// Mitsubishi GX Works2 project: CV_B01-20251214_0   PLC: Q03UDV

TYPE DInput : STRUCT
  In_Power : BOOL;  (* 输入电源 *)
  X01_1 : BOOL;  (* X01_1 *)
  B01_Emergency_Stop_Circuit1 : BOOL;  (* BO1急停回路1 *)
  B01_Emergency_Stop_Circuit2 : BOOL;  (* BO1急停回路2 *)
  B01_Grating_Circuit1 : BOOL;  (* BO1光栅回路1 *)
  B01_Grating_Circuit2 : BOOL;  (* BO1光栅回路2 *)
  B01_Safety_Door_Circuit1 : BOOL;  (* BO1安全门回路1 *)
  B01_Safety_Door_Circuit2 : BOOL;  (* BO1安全门回路2 *)
  AO1Safety_Circuit1 : BOOL;  (* AO1急停回路1 *)
  AO1Safety_Circuit2 : BOOL;  (* AO1急停回路2 *)
  B02_Emergency_Stop_Circuit1 : BOOL;  (* BO2急停回路1 *)
  B02_Emergency_Stop_Circuit2 : BOOL;  (* BO2急停回路2 *)
  B02_Grating_Circuit1 : BOOL;  (* BO2光栅回路1 *)
  B02_Grating_Circuit2 : BOOL;  (* BO2光栅回路2 *)
  B02_Safety_Door_Circuit1 : BOOL;  (* BO2安全门回路1 *)
  B02_Safety_Door_Circuit2 : BOOL;  (* BO2安全门回路2 *)
  Manual_Auto : BOOL;  (* 手动自动 *)
  Single_OnLine : BOOL;  (* 单机联机 *)
  X02_2 : BOOL;  (* X02_2 *)
  Admin : BOOL;  (* 管理者 *)
  Alarm_Reset : BOOL;  (* 故障复位 *)
  Ready_Button : BOOL;  (* 就绪按钮 *)
  Start_Button : BOOL;  (* 启动按钮 *)
  Pause_Button : BOOL;  (* 暂停按钮 *)
  Lamp_Check : BOOL;  (* 灯光检查按钮 *)
  X09_2 : BOOL;  (* X09_2 *)
  Operational_Ready1 : BOOL;  (* 运行准备01 *)
  Operational_Ready2 : BOOL;  (* 运行准备02 *)
  Operational_Ready11 : BOOL;  (* 运行准备11 *)
  Operational_Ready12 : BOOL;  (* 运行准备12 *)
  Air_Error : BOOL;  (* 柜机空调故障 *)
  X0F_2 : BOOL;  (* X0F_2 *)
  CV01顶升上限检测 : BOOL;  (* CV01顶升上限检测 *)
  CV01顶升下限检测 : BOOL;  (* CV01顶升下限检测 *)
  CV01顶升故障检测 : BOOL;  (* CV01顶升故障检测 *)
  CV01顶升电源检测 : BOOL;  (* CV01顶升电源检测 *)
  CV01物料停止检测 : BOOL;  (* CV01物料停止检测 *)
  X05_3 : BOOL;  (* X05_3 *)
  CV01伸缩中位检测1 : BOOL;  (* CV01伸缩中位检测1 *)
  CV01伸缩中位检测2 : BOOL;  (* CV01伸缩中位检测2 *)
  CV01伸缩极限检测 : BOOL;  (* CV01伸缩极限检测 *)
  CV01伸缩电源检测 : BOOL;  (* CV01伸缩电源检测 *)
  CV01AGV物料检测 : BOOL;  (* CV01AGV物料检测 *)
  CV01AGV本体检测1 : BOOL;  (* CV01AGV本体检测1 *)
  CV01AGV本体检测2 : BOOL;  (* CV01AGV本体检测2 *)
  CV01超宽检测1 : BOOL;  (* CV01超宽检测1 *)
  CV01超宽检测2 : BOOL;  (* CV01超宽检测2 *)
  CV01超高检测 : BOOL;  (* CV01超高检测 *)
  Bx03顶升上限检测 : BOOL;  (* Bx03顶升上限检测 *)
  Bx03顶升下限检测 : BOOL;  (* Bx03顶升下限检测 *)
  Bx03顶升故障检测 : BOOL;  (* Bx03顶升故障检测 *)
  Bx03顶升电源检测 : BOOL;  (* Bx03顶升电源检测 *)
  Bx03物料停止检测 : BOOL;  (* Bx03物料停止检测 *)
  Bx03物料减速检测 : BOOL;  (* Bx03物料减速检测 *)
  CV02伸缩中位检测1 : BOOL;  (* Bx03伸缩中位检测1 *)
  CV02伸缩中位检测2 : BOOL;  (* Bx03伸缩中位检测2 *)
  CV02伸缩极限检测 : BOOL;  (* Bx03伸缩极限检测 *)
  Bx03伸缩电源检测 : BOOL;  (* Bx03伸缩电源检测 *)
  Bx03AGV物料检测 : BOOL;  (* Bx03AGV物料检测 *)
  Bx03AGV本体检测1 : BOOL;  (* Bx03AGV本体检测1 *)
  Bx03AGV本体检测2 : BOOL;  (* Bx03AGV本体检测2 *)
  X0D_4 : BOOL;  (* X0D_4 *)
  X0E_4 : BOOL;  (* X0E_4 *)
  X0F_4 : BOOL;  (* X0F_4 *)
  Bx02顶升上限检测 : BOOL;  (* Bx02顶升上限检测 *)
  Bx02顶升下限检测 : BOOL;  (* Bx02顶升下限检测 *)
  Bx02顶升故障检测 : BOOL;  (* Bx02顶升故障检测 *)
  Bx02顶升电源检测 : BOOL;  (* Bx02顶升电源检测 *)
  Bx02物料到位检测 : BOOL;  (* Bx02物料到位检测 *)
  Bx02物料减速检测 : BOOL;  (* Bx02物料减速检测 *)
  Bx02输送故障检测 : BOOL;  (* Bx02输送故障检测 *)
  Bx02输送电源检测 : BOOL;  (* Bx02输送电源检测 *)
  Bx04顶升上限检测 : BOOL;  (* Bx04顶升上限检测 *)
  Bx04顶升下限检测 : BOOL;  (* Bx04顶升下限检测 *)
  Bx04顶升故障检测 : BOOL;  (* Bx04顶升故障检测 *)
  Bx04顶升电源检测 : BOOL;  (* Bx04顶升电源检测 *)
  Bx04物料到位检测 : BOOL;  (* Bx04物料到位检测 *)
  X0D_5 : BOOL;  (* X0D_5 *)
  Bx04输送故障检测 : BOOL;  (* Bx04输送故障检测 *)
  Bx04输送电源检测 : BOOL;  (* Bx04输送电源检测 *)
  AGV侧安全光栅输入信号1 : BOOL;  (* AGV侧安全光栅输入信号1 *)
  AGV侧安全光栅输入信号2 : BOOL;  (* AGV侧安全光栅输入信号2 *)
  AGV侧安全光栅输入信号11 : BOOL;  (* AGV侧安全光栅输入信号11 *)
  AGV侧安全光栅输入信号12 : BOOL;  (* AGV侧安全光栅输入信号12 *)
  CV_IN侧安全光栅输入信号1 : BOOL;  (* CV_IN侧安全光栅输入信号1 *)
  CV_IN侧安全光栅输入信号2 : BOOL;  (* CV_IN侧安全光栅输入信号2 *)
  CV_Out侧安全光栅输入信号1 : BOOL;  (* CV_Out侧安全光栅输入信号1 *)
  CV_Out侧安全光栅输入信号2 : BOOL;  (* CV_Out侧安全光栅输入信号2 *)
  X08_6 : BOOL;  (* X08_6 *)
  X09_6 : BOOL;  (* X09_6 *)
  安全门1输入信号1 : BOOL;  (* 安全门1输入信号1 *)
  安全门1输入信号2 : BOOL;  (* 安全门1输入信号2 *)
  解锁1安全门 : BOOL;  (* 解锁1安全门 *)
  X0D_6 : BOOL;  (* X0D_6 *)
  X0E_6 : BOOL;  (* X0E_6 *)
  X0F_6 : BOOL;  (* X0F_6 *)
  Photonic1_output1 : BOOL;  (* Photonic1_output1 *)
  Photonic1_output2 : BOOL;  (* Photonic1_output2 *)
  Photonic1_output3 : BOOL;  (* Photonic1_output3 *)
  Photonic1_output4 : BOOL;  (* Photonic1_output4 *)
  Photonic1_Go : BOOL;  (* Photonic1_Go *)
  X05_7 : BOOL;  (* X05_7 *)
  Photonic2_output1 : BOOL;  (* Photonic2_output1 *)
  Photonic2_output2 : BOOL;  (* Photonic2_output2 *)
  Photonic2_output3 : BOOL;  (* Photonic2_output3 *)
  Photonic2_output4 : BOOL;  (* Photonic2_output4 *)
  Photonic2_Go : BOOL;  (* Photonic2_Go *)
  X0B_7 : BOOL;  (* X0B_7 *)
  Photonic3_output1 : BOOL;  (* Photonic3_output1 *)
  Photonic3_output2 : BOOL;  (* Photonic3_output2 *)
  Photonic3_output3 : BOOL;  (* Photonic3_output3 *)
  Photonic3_output4 : BOOL;  (* Photonic3_output4 *)
  Photonic3_Go : BOOL;  (* Photonic3_Go *)
  X01_8 : BOOL;  (* X01_8 *)
  Photonic4_output1 : BOOL;  (* Photonic4_output1 *)
  Photonic4_output2 : BOOL;  (* Photonic4_output2 *)
  Photonic4_output3 : BOOL;  (* Photonic4_output3 *)
  Photonic4_output4 : BOOL;  (* Photonic4_output4 *)
  Photonic4_Go : BOOL;  (* Photonic4_Go *)
  X07_8 : BOOL;  (* X07_8 *)
  X08_8 : BOOL;  (* X08_8 *)
  X09_8 : BOOL;  (* X09_8 *)
  X0A_8 : BOOL;  (* X0A_8 *)
  X0B_8 : BOOL;  (* X0B_8 *)
  X0C_8 : BOOL;  (* X0C_8 *)
  X0D_8 : BOOL;  (* X0D_8 *)
  X0E_8 : BOOL;  (* X0E_8 *)
  X0F_8 : BOOL;  (* X0F_8 *)
END_STRUCT END_TYPE

TYPE DOutput : STRUCT
  Pole_Light_R : BOOL;  (* 柜体灯_红 *)
  Pole_Light_Y : BOOL;  (* 柜体灯_黄 *)
  Pole_Light_G : BOOL;  (* 柜体灯_绿 *)
  HA01_Sound1 : BOOL;  (* 蜂鸣器通道1 *)
  HA01_Sound2 : BOOL;  (* 蜂鸣器通道2 *)
  HA01_Sound3 : BOOL;  (* 蜂鸣器通道3 *)
  HA01_Sound4 : BOOL;  (* 蜂鸣器通道4 *)
  Y07_1 : BOOL;  (* Y07_1 *)
  Ready_Button_Indicator_Light : BOOL;  (* 就绪按钮灯 *)
  Start_Button_Indicator_Light : BOOL;  (* 启动按钮灯 *)
  Pause_Button_Indicator_Light : BOOL;  (* 暂停按钮灯 *)
  Y0B_1 : BOOL;  (* Y0B_1 *)
  Y0C_1 : BOOL;  (* Y0C_1 *)
  Y0D_1 : BOOL;  (* Y0D_1 *)
  SafetyDoor_Indicator_Light : BOOL;  (* Lock the Safety Door *)
  Unlock_SafetyDoor : BOOL;  (* 解锁安全门 *)
  CV1_JackingUP_Fork_Run : BOOL;  (* Bx01顶升正转运行 *)
  CV1_JackingDown_Fork_Run : BOOL;  (* Bx01顶升反转运行 *)
  CV1_Jacking_Fork_Reset : BOOL;  (* Bx01顶升故障复位 *)
  Y03_2 : BOOL;  (* Y03_2 *)
  Grat1_Warning_Light_R : BOOL;  (* 光栅1警示灯_红 *)
  Grat1_Warning_Light_G : BOOL;  (* 光栅1警示灯_绿 *)
  CV1_JackingUP_Run : BOOL;  (* Bx02顶升正转运行 *)
  CV1_JackingDown_Run : BOOL;  (* Bx02顶升反转运行 *)
  CV1_Jacking_Reset : BOOL;  (* Bx02顶升故障复位 *)
  Y09_2 : BOOL;  (* Y09_2 *)
  CV1_ConveyingIN_Run : BOOL;  (* Bx02输送正转运行 *)
  CV1_ConveyingOut_Run : BOOL;  (* Bx02输送反转运行 *)
  CV1_Conveying_SpeedA : BOOL;  (* Bx02输送速度A *)
  CV1_Conveying_SpeedB : BOOL;  (* Bx02输送速度B *)
  CV1_Conveying_Reset : BOOL;  (* Bx02输送故障复位 *)
  Y0F_2 : BOOL;  (* Y0F_2 *)
  CV2_JackingUP_Fork_Run : BOOL;  (* Bx03顶升正转运行 *)
  CV2_JackingDown_Fork_Run : BOOL;  (* Bx03顶升反转运行 *)
  CV2_Jacking_Fork_Reset : BOOL;  (* Bx03顶升故障复位 *)
  Y03_3 : BOOL;  (* Y03_3 *)
  Grat2_Warning_Light_R : BOOL;  (* 光栅2警示灯_红 *)
  Grat2_Warning_Light_G : BOOL;  (* 光栅2警示灯_绿 *)
  CV2_JackingUP_Run : BOOL;  (* Bx04顶升正转运行 *)
  CV2_JackingDown_Run : BOOL;  (* Bx04顶升反转运行 *)
  CV2_Jacking_Reset : BOOL;  (* Bx04顶升故障复位 *)
  Y09_3 : BOOL;  (* Y09_3 *)
  CV2_ConveyingIN_Run : BOOL;  (* Bx04输送正转运行 *)
  CV2_ConveyingOut_Run : BOOL;  (* Bx04输送反转运行 *)
  CV2_Conveying_SpeedA : BOOL;  (* Bx04输送速度A *)
  CV2_Conveying_SpeedB : BOOL;  (* Bx04输送速度B *)
  CV2_Conveying_Reset : BOOL;  (* Bx04输送故障复位 *)
  Y0F_3 : BOOL;  (* Y0F_3 *)
  Photonic1_Input1 : BOOL;  (* Photonic1_Input1 *)
  Photonic1_Input2 : BOOL;  (* Photonic1_Input2 *)
  Photonic1_Input3 : BOOL;  (* Photonic1_Input3 *)
  Photonic1_Input4 : BOOL;  (* Photonic1_Input4 *)
  Photonic2_Input1 : BOOL;  (* Photonic2_Input1 *)
  Photonic2_Input2 : BOOL;  (* Photonic2_Input2 *)
  Photonic2_Input3 : BOOL;  (* Photonic2_Input3 *)
  Photonic2_Input4 : BOOL;  (* Photonic2_Input4 *)
  Photonic3_Input1 : BOOL;  (* Photonic3_Input1 *)
  Photonic3_Input2 : BOOL;  (* Photonic3_Input2 *)
  Photonic3_Input3 : BOOL;  (* Photonic3_Input3 *)
  Photonic3_Input4 : BOOL;  (* Photonic3_Input4 *)
  Photonic4_Input1 : BOOL;  (* Photonic4_Input1 *)
  Photonic4_Input2 : BOOL;  (* Photonic4_Input2 *)
  Photonic4_Input3 : BOOL;  (* Photonic4_Input3 *)
  Photonic4_Input4 : BOOL;  (* Photonic4_Input4 *)
  Y00_5 : BOOL;  (* Y00_5 *)
  Y01_5 : BOOL;  (* Y01_5 *)
  Y02_5 : BOOL;  (* Y02_5 *)
  Y03_5 : BOOL;  (* Y03_5 *)
  Y04_5 : BOOL;  (* Y04_5 *)
  Y05_5 : BOOL;  (* Y05_5 *)
  Invalid_CV_IN_Grat1 : BOOL;  (* 屏蔽CV_IN侧光栅信号1 *)
  Invalid_CV_IN_Grat2 : BOOL;  (* 屏蔽CV_IN侧光栅信号2 *)
  Y08_5 : BOOL;  (* Y08_5 *)
  Invalid_CV_OUT_Grat1 : BOOL;  (* 屏蔽CV_OUT侧光栅信号1 *)
  Invalid_CV_OUT_Grat2 : BOOL;  (* 屏蔽CV_OUT侧光栅信号2 *)
  Y0B_5 : BOOL;  (* Y0B_5 *)
  Invalid_SafetyDoor1 : BOOL;  (* 屏蔽安全门信号1 *)
  Invalid_SafetyDoor2 : BOOL;  (* 屏蔽安全门信号2 *)
  Y0E_5 : BOOL;  (* Y0E_5 *)
  Y0F_5 : BOOL;  (* Y0F_5 *)
END_STRUCT END_TYPE

TYPE Deliver_In : STRUCT
  货叉位置物料检测 : BOOL;  (* 货叉位置物料检测 *)
  入库口减速检测 : BOOL;  (* 入库口减速检测 *)
  入库口物料检测 : BOOL;  (* 入库口物料检测 *)
  入库口顶升上限检测 : BOOL;  (* 入库口顶升上限检测 *)
  入库口顶升下限检测 : BOOL;  (* 入库口顶升下限检测 *)
  AGV_Stop_Status : BOOL;  (* AGV停止 *)
  AGV_Go : BOOL;  (* AGV就绪 *)
  AGV物料探测 : BOOL;  (* AGV物料探测 *)
  货叉顶升上限检测 : BOOL;  (* 货叉顶升上限检测 *)
  货叉顶升下限检测 : BOOL;  (* 货叉顶升下限检测 *)
  货叉伸出到位 : BOOL;  (* 货叉伸出到位 *)
  货叉缩回到位 : BOOL;  (* 货叉缩回到位 *)
  输送线控制 : BOOL;  (* 输送线控制 *)
  输送线低速控制 : BOOL;  (* 输送线低速控制 *)
  入库口顶升上升控制 : BOOL;  (* 入库口顶升上升控制 *)
  入库口顶升下降控制 : BOOL;  (* 入库口顶升下降控制 *)
  货叉顶升上升控制 : BOOL;  (* 货叉顶升上升控制 *)
  货叉顶升下降控制 : BOOL;  (* 货叉顶升下降控制 *)
  货叉伸出控制 : BOOL;  (* 货叉伸出控制 *)
  货叉缩回控制 : BOOL;  (* 货叉缩回控制 *)
  Current_Task_Status : INT;  (* 当前任务状态 *)
  Step1 : INT;  (* Step1 *)
  Current_TaskID : DWORD;  (* 当前任务ID *)
  Task_ID : DWORD;  (* Task_ID *)
  AGV进入中 : BOOL;  (* AGV进入中 *)
  AGV本体检测 : BOOL;  (* AGV本体检测 *)
  AGV放行 : BOOL;  (* AGV放行 *)
END_STRUCT END_TYPE

TYPE Deliver_Out : STRUCT
  Task_ID : DWORD;  (* Task_ID *)
  货叉位置物料检测 : BOOL;  (* 货叉位置物料检测 *)
  货叉位置减速检测 : BOOL;  (* 货叉位置减速检测 *)
  出库口物料检测 : BOOL;  (* 出库口物料检测 *)
  出库口顶升上限检测 : BOOL;  (* 出库口顶升上限检测 *)
  出库口顶升下限检测 : BOOL;  (* 出库口顶升下限检测 *)
  AGV_Stop_Status : BOOL;  (* AGV停止 *)
  AGV_Go : BOOL;  (* AGV就绪 *)
  AGV物料探测 : BOOL;  (* AGV物料探测 *)
  货叉顶升上限检测 : BOOL;  (* 货叉顶升上限检测 *)
  货叉顶升下限检测 : BOOL;  (* 货叉顶升下限检测 *)
  货叉伸出到位 : BOOL;  (* 货叉伸出到位 *)
  货叉缩回到位 : BOOL;  (* 货叉缩回到位 *)
  输送线控制 : BOOL;  (* 输送线控制 *)
  输送线低速控制 : BOOL;  (* 输送线低速控制 *)
  出库口顶升上升控制 : BOOL;  (* 出库口顶升上升控制 *)
  出库口顶升下降控制 : BOOL;  (* 出库口顶升下降控制 *)
  货叉顶升上升控制 : BOOL;  (* 货叉顶升上升控制 *)
  货叉顶升下降控制 : BOOL;  (* 货叉顶升下降控制 *)
  货叉伸出控制 : BOOL;  (* 货叉伸出控制 *)
  货叉缩回控制 : BOOL;  (* 货叉缩回控制 *)
  Current_TaskID : DWORD;  (* 当前任务ID *)
  Current_Task_Status : INT;  (* 当前任务状态 *)
  Step1 : INT;  (* Step1 *)
  AGV放行 : BOOL;  (* AGV放行 *)
  AGVl离开中 : BOOL;  (* AGVl离开中 *)
  AGV本体检测 : BOOL;  (* AGV本体检测 *)
END_STRUCT END_TYPE

TYPE manual_Data : STRUCT
  手动入库货叉上升 : BOOL;  (* 手动入库货叉上升 *)
  手动入库货叉下降 : BOOL;  (* 手动入库货叉下降 *)
  手动入库货叉伸出 : BOOL;  (* 手动入库货叉伸出 *)
  手动入库货叉缩回 : BOOL;  (* 手动入库货叉缩回 *)
  手动入库输送线运转 : BOOL;  (* 手动入库输送线运转 *)
  手动入库台上升 : BOOL;  (* 手动入库台上升 *)
  手动入库台下降 : BOOL;  (* 手动入库台下降 *)
  手动出库货叉上升 : BOOL;  (* 手动出库货叉上升 *)
  手动出库货叉下降 : BOOL;  (* 手动出库货叉下降 *)
  手动出库货叉伸出 : BOOL;  (* 手动出库货叉伸出 *)
  手动出库货叉缩回 : BOOL;  (* 手动出库货叉缩回 *)
  手动出库输送线运转 : BOOL;  (* 手动出库输送线运转 *)
  手动出库台上升 : BOOL;  (* 手动出库台上升 *)
  手动出库台下降 : BOOL;  (* 手动出库台下降 *)
  手动入库输送线反转 : BOOL;  (* 手动入库输送线反转 *)
  手动出库输送线反转 : BOOL;  (* 手动出库输送线反转 *)
  自动入库货叉伸出 : BOOL;  (* 自动入库货叉伸出 *)
  自动入库货叉缩回 : BOOL;  (* 自动入库货叉缩回 *)
  自动出库货叉伸出 : BOOL;  (* 自动出库货叉伸出 *)
  自动出库货叉缩回 : BOOL;  (* 自动出库货叉缩回 *)
END_STRUCT END_TYPE

TYPE HMI : STRUCT
  自动联机模式 : BOOL;  (* 自动联机模式 *)
  自动单机模式 : BOOL;  (* 自动单机模式 *)
  手动模式 : BOOL;  (* 手动模式 *)
  维修模式 : BOOL;  (* 维修模式 *)
  Alarm_Reset : BOOL;  (* 报警复位 *)
  Invalid_CV_IN_Grat : BOOL;  (* 入库侧光栅屏蔽 *)
  Invalid_CV_OUT_Grat : BOOL;  (* 出库侧光栅屏蔽 *)
  Invalid_SafetyDoor : BOOL;  (* 安全门屏蔽 *)
  Invalid_AGV_IN_Grat : BOOL;  (* AGV入侧光栅屏蔽 *)
  Invalid_AGV_OUT_Grat : BOOL;  (* AGV出侧光栅屏蔽 *)
END_STRUCT END_TYPE

TYPE Sew_Control_Bit : STRUCT
  Enable_Emergency_Stop : BOOL;  (* 使能紧急停止 *)
  Enable_Application_Stop : BOOL;  (* 使能应用停止 *)
  预留1 : BOOL;  (* 预留1 *)
  Brake_Open : BOOL;  (* 制动器释放 *)
  Forward_Jog : BOOL;  (* 正点动 *)
  Reverse_Jog : BOOL;  (* 负点动 *)
  接收相对位置 : BOOL;  (* 接收相对位置 *)
  Ramp_Bus_StartStop : BOOL;  (* 随总线斜波启动停止 *)
  Alarm_Reset : BOOL;  (* 故障复位 *)
  预留2 : BOOL;  (* 预留2 *)
  激活驱动机构2 : BOOL;  (* 激活驱动机构2 *)
  预留3 : BOOL;  (* 预留3 *)
  禁用软件限位开关 : BOOL;  (* 禁用软件限位开关 *)
  激活输出级锁定 : BOOL;  (* 激活输出级锁定 *)
  激活待机运行 : BOOL;  (* 激活待机运行 *)
  HandshakeIn : BOOL;  (* HandshakeIn *)
END_STRUCT END_TYPE

TYPE Sew_Read : STRUCT
  Status_Character : INT;  (* 状态字 *)
  Actual_Speed : INT;  (* 实际速度 *)
  Main_Status_Fault : WORD;  (* 状态主故障 *)
  Actual_Torque : INT;  (* 实际扭矩 *)
  Digital_Input_Port : INT;  (* 数字输入端 *)
  Actual_Mode : INT;  (* 实际应用模式 *)
  Actual_Position : DINT;  (* 实际位置 *)
END_STRUCT END_TYPE

TYPE Sew_Status_Bit : STRUCT
  Ready_To_Run : BOOL;  (* 运行就绪 *)
  STO非活跃 : BOOL;  (* STO非活跃 *)
  输出级已使能 : BOOL;  (* 输出级已使能 *)
  制动器已打开 : BOOL;  (* 制动器已打开 *)
  电机旋转 : BOOL;  (* 电机旋转 *)
  Homed : BOOL;  (* 激活的驱动装置已寻参 *)
  已应用新的相对位置 : BOOL;  (* 已应用新的相对位置 *)
  Position_Arrive : BOOL;  (* 信息已就位激活 *)
  Error : BOOL;  (* 故障 *)
  警告 : BOOL;  (* 警告 *)
  驱动机构2激活 : BOOL;  (* 驱动机构2激活 *)
  消息额定_实际速度比较激活 : BOOL;  (* 消息额定_实际速度比较激活 *)
  软件限位开关非活跃 : BOOL;  (* 软件限位开关非活跃 *)
  预留 : BOOL;  (* 预留 *)
  待机运行激活 : BOOL;  (* 待机运行激活 *)
  HandshakeOut : BOOL;  (* HandshakeOut *)
END_STRUCT END_TYPE

TYPE Sew_Write : STRUCT
  Control_Character : INT;  (* 控制字 *)
  Rated_Speed : INT;  (* 额定速度 *)
  Acceleration : INT;  (* 加速度 *)
  Deceleration : INT;  (* 减速度 *)
  Virtual_Input_Port : INT;  (* 虚拟输入端 *)
  Set_Mode : INT;  (* 设定应用模式 *)
  Target_Position : DINT;  (* 目标位置 *)
END_STRUCT END_TYPE

TYPE parameter : STRUCT
  CV1_Fork_Speed_Set : INT;  (* 入库货叉速度设置 *)
  CV2_Fork_Speed_Set : INT;  (* 出库货叉速度设置 *)
  CV1_Fork_Position_Set : DINT;  (* 入库货叉位置设置 *)
  CV2_Fork_Position_Set : DINT;  (* 出库货叉位置设置 *)
  CV1_Fork_Acceleration_Set : INT;  (* 入库货叉加速度 *)
  CV1_Fork_Deceleration_Set : INT;  (* 入库货叉减速度 *)
  CV2_Fork_Acceleration_Set : INT;  (* 出库货叉加速度 *)
  CV2_Fork_Deceleration_Set : INT;  (* 出库货叉减速度 *)
  CV1_Fork_Pos_Offset : DINT;  (* 入库货叉位置偏移设置 *)
  CV2_Fork_Pos_Offset : DINT;  (* 出库货叉位置偏移设置 *)
END_STRUCT END_TYPE

TYPE Master_R : STRUCT
  Heartbeat : INT;  (* 心跳检测 *)
  Current_Mode : INT;  (* 当前模式 *)
  Device_Status : INT;  (* 设备状态 *)
  CV1_Task_Status : INT;  (* 入库线_任务状态 *)
  CV1_AGVPick_Goods_Done : INT;  (* 站台1001AGV取货完成 *)
  Stacker_PickingGoods_Status : INT;  (* 堆垛机允许取货1002 *)
  CV2_Task_Status : INT;  (* 出库线_任务状态 *)
  Error_Code : INT;  (* 错误码 *)
  CV1_Current_TaskID : DWORD;  (* 站台1002任务ID *)
  CV2_Current_TaskID : DWORD;  (* 站台1003任务ID *)
  Stacker_UnloadGoods_Status : INT;  (* 堆垛机允许放货1004 *)
  CV1_Current_RFID : STRING[12];  (* 站台1001RFID读取值 *)
  CV2_Current_RFID : STRING[12];  (* 站台1003RIFD读取值 *)
  Spare1 : INT;  (* 备用1 *)
  Spare2 : INT;  (* 备用2 *)
  Spare3 : INT;  (* 备用3 *)
  Spare4 : INT;  (* 备用4 *)
  Spare5 : INT;  (* 备用5 *)
END_STRUCT END_TYPE

TYPE Master_W : STRUCT
  货叉站台任务ID : DWORD;  (* 货叉站台任务ID *)
  Heartbeat : INT;  (* 心跳检测 *)
  入库站台堆垛机取货完成 : INT;  (* 1002入库站台堆垛机取货完成 *)
  出库站台任务ID : DWORD;  (* 1004出库站台任务ID *)
  允许出料到AGV : INT;  (* 1003允许出料到AGV *)
  出库口空托余料不足报警 : INT;  (* 出库口空托余料不足报警 *)
  入库RFID物料不匹配报警 : INT;  (* 入库RFID物料不匹配报警 *)
  备用0 : INT;  (* 备用0 *)
  备用10 : INT;  (* 备用10 *)
  备用1 : INT;  (* 备用1 *)
  备用2 : INT;  (* 备用2 *)
  备用3 : INT;  (* 备用3 *)
  备用4 : INT;  (* 备用4 *)
  备用5 : INT;  (* 备用5 *)
  备用6 : INT;  (* 备用6 *)
  备用7 : INT;  (* 备用7 *)
  备用8 : INT;  (* 备用8 *)
  备用9 : INT;  (* 备用9 *)
END_STRUCT END_TYPE

TYPE CCLink_R : STRUCT
  Heartbeat : INT;  (* 心跳检测 *)
  Current_Mode : INT;  (* 当前模式 *)
  Device_Status : INT;  (* 设备状态 *)
  Error_Code : INT;  (* 错误码 *)
  CV1_Task_Status : INT;  (* 入库线_任务状态 *)
  CV1_AGVPick_Goods_Done : INT;  (* 站台1001AGV取货完成 *)
  CV1_Current_TaskID : DWORD;  (* 站台1002任务ID *)
  Stacker_PickingGoods_Status : INT;  (* 堆垛机允许取货1002 *)
  CV2_Task_Status : INT;  (* 出库线_任务状态 *)
  CV2_Current_TaskID : DWORD;  (* 站台1003任务ID *)
  Stacker_UnloadGoods_Status : INT;  (* 堆垛机允许放货1004 *)
  CV1_Current_RFID : STRING[12];  (* 站台1001RFID读取值 *)
  CV2_Current_RFID : STRING[12];  (* 站台1003RIFD读取值 *)
  CV1_Step : INT;  (* 入库流程字 *)
  CV2_Step : INT;  (* 出库流程字 *)
  CV2_AGVReleaseGoods_Done : INT;  (* 出库AGV放货完成 *)
  CV2_AGVPurpose : INT;  (* 出库AGV目的地 *)
  CV1_Fork_Current_Pos : INT;  (* 入库货叉位置 *)
  CV2_Fork_Current_Pos : INT;  (* 出库货叉位置 *)
  Spare7 : INT;  (* 备用7 *)
  Spare8 : INT;  (* 备用8 *)
  Spare9 : INT;  (* 备用9 *)
  Spare10 : INT;  (* 备用10 *)
  Spare11 : INT;  (* 备用11 *)
  Spare12 : INT;  (* 备用12 *)
  Spare13 : INT;  (* 备用13 *)
  Spare14 : INT;  (* 备用14 *)
  Spare15 : INT;  (* 备用15 *)
  Spare16 : INT;  (* 备用16 *)
  Spare17 : INT;  (* 备用17 *)
  Spare18 : INT;  (* 备用18 *)
  Spare19 : INT;  (* 备用19 *)
  Spare20 : INT;  (* 备用20 *)
  Spare21 : INT;  (* 备用21 *)
END_STRUCT END_TYPE

TYPE CCLink_W : STRUCT
  Heartbeat : INT;  (* 心跳检测 *)
  CV1_TaskID : DWORD;  (* 货叉站台任务ID *)
  CV1_Stacker_Pick_Goods_Done : INT;  (* 1002入库站台堆垛机取货完成 *)
  CV2_TaskID : DWORD;  (* 1004出库站台任务ID *)
  CV2_Allow_GoodsToAGV : INT;  (* 1003允许出料到AGV *)
  CV1_RFID_Alarm : INT;  (* 入库口RFID报警 *)
  CV2_RFID_Alarm : INT;  (* 出库口RFID报警 *)
  Spare0 : INT;  (* 备用0 *)
  Spare1 : INT;  (* 备用1 *)
  A01_Mode : INT;  (* A01_Mode *)
  Spare2 : INT;  (* 备用2 *)
  Spare3 : INT;  (* 备用3 *)
  Spare4 : INT;  (* 备用4 *)
  Spare5 : INT;  (* 备用5 *)
  Spare6 : INT;  (* 备用6 *)
  Spare7 : INT;  (* 备用7 *)
  Spare8 : INT;  (* 备用8 *)
  Spare9 : INT;  (* 备用9 *)
  Spare10 : INT;  (* 备用10 *)
  Spare11 : INT;  (* 备用11 *)
  Spare12 : INT;  (* 备用12 *)
  Spare13 : INT;  (* 备用13 *)
  Spare14 : INT;  (* 备用14 *)
  Spare15 : INT;  (* 备用15 *)
  Spare16 : INT;  (* 备用16 *)
  Spare17 : INT;  (* 备用17 *)
  Spare18 : INT;  (* 备用18 *)
  Spare19 : INT;  (* 备用19 *)
  Spare20 : INT;  (* 备用20 *)
  Spare32_48 : ARRAY [0..15] OF INT;  (* 备用32_48 *)
END_STRUCT END_TYPE

TYPE CCLink_W_Control_Bit : STRUCT
  Alarm_Reset : BOOL;  (* 故障复位 *)
  Stacker_Picking_Goods_Mark : BOOL;  (* 取货中 *)
  Stacker_Unload_Goodsv_Mark : BOOL;  (* 放货中 *)
  Spare3 : BOOL;  (* 备用3 *)
  Spare4 : BOOL;  (* 备用4 *)
  Spare5 : BOOL;  (* 备用5 *)
  Spare6 : BOOL;  (* 备用6 *)
  Spare7 : BOOL;  (* 备用7 *)
  Spare8 : BOOL;  (* 备用8 *)
  Spare9 : BOOL;  (* 备用9 *)
END_STRUCT END_TYPE

TYPE CCLink_R_Status_Bit : STRUCT
  入库货叉台物料检测 : BOOL;  (* 入库货叉台物料检测 *)
  入库台减速检测 : BOOL;  (* 入库台减速检测 *)
  入库台物料检测 : BOOL;  (* 入库台物料检测 *)
  出库货叉台物料检测 : BOOL;  (* 出库货叉台物料检测 *)
  出库货叉台减速检测 : BOOL;  (* 出库货叉台减速检测 *)
  出库台物料检测 : BOOL;  (* 出库台物料检测 *)
  入库货叉上限检测 : BOOL;  (* 入库货叉上限检测 *)
  入库货叉下限检测 : BOOL;  (* 入库货叉下限检测 *)
  入库台上限检测 : BOOL;  (* 入库台上限检测 *)
  入库台下限检测 : BOOL;  (* 入库台下限检测 *)
  出库货叉上限检测 : BOOL;  (* 出库货叉上限检测 *)
  出库货叉下限检测 : BOOL;  (* 出库货叉下限检测 *)
  出库台上限检测 : BOOL;  (* 出库台上限检测 *)
  出库台下限检测 : BOOL;  (* 出库台下限检测 *)
  入库超宽检测1 : BOOL;  (* 入库超宽检测1 *)
  入库超宽检测2 : BOOL;  (* 入库超宽检测2 *)
  入库超高检测 : BOOL;  (* 入库超高检测 *)
  入库坍塌检测 : BOOL;  (* 入库坍塌检测 *)
  入库光栅 : BOOL;  (* 入库光栅 *)
  出库光栅 : BOOL;  (* 出库光栅 *)
  AGV入光栅 : BOOL;  (* AGV入光栅 *)
  AGV出光栅 : BOOL;  (* AGV出光栅 *)
  安全门状态 : BOOL;  (* 安全门状态 *)
  入库agv本体检测 : BOOL;  (* 入库agv本体检测 *)
  入库agv物料检测 : BOOL;  (* 入库agv物料检测 *)
  出库agv本体检测 : BOOL;  (* 出库agv本体检测 *)
  出库agv物料检测 : BOOL;  (* 出库agv物料检测 *)
  入库货叉极限 : BOOL;  (* 入库货叉极限 *)
  入库货叉原点 : BOOL;  (* 入库货叉原点 *)
  出库库货叉极限 : BOOL;  (* 出库库货叉极限 *)
  出库货叉原点 : BOOL;  (* 出库货叉原点 *)
  备用1 : BOOL;  (* 备用1 *)
  备用2 : BOOL;  (* 备用2 *)
  备用3 : BOOL;  (* 备用3 *)
  备用4 : BOOL;  (* 备用4 *)
  备用5 : BOOL;  (* 备用5 *)
  备用6 : BOOL;  (* 备用6 *)
  备用7 : BOOL;  (* 备用7 *)
  备用8 : BOOL;  (* 备用8 *)
  备用9 : BOOL;  (* 备用9 *)
END_STRUCT END_TYPE

TYPE RFID : STRUCT
  Q1 : STRING[2];
  Q2 : STRING[2];
  Q3 : STRING[2];
  Q4 : STRING[2];
  Q5 : STRING[2];
  Q6 : STRING[2];
END_STRUCT END_TYPE

// global labels: Global1
VAR_GLOBAL
  DInput : DInput;
  DOutput : DOutput;
  E_Stop : BOOL;
  Alarm_Code AT D1005 : INT;  (* 错误码 *)
  Mode AT D1008 : INT;
  Deliver_In : Deliver_In;
  Deliver_Out : Deliver_Out;
  Manual : manual_Data;
  Device_Station : BOOL;  (* 设备静止中 *)
  OnLine_Mode AT M502 : BOOL;  (* 自动联机模式状态 *)
  Single_Mode AT M503 : BOOL;  (* 自动单机模式状态 *)
  Manual_Mode AT M504 : BOOL;  (* 手动模式状态 *)
  Maintenance_Mode AT M505 : BOOL;  (* 维修模式状态 *)
  Language_Switch AT M700 : BOOL;  (* 语言切换 *)
  Language AT D5030 : INT;  (* 语言显示 *)
  Password AT D5032 : INT;  (* 密码权限 *)
  HMI : HMI;  (* HMI *)
  parameter : parameter;
  Master_R : Master_R;
  Master_W : Master_W;
  SingleID_Cv1 AT D1200 : DWORD;  (* 单机入库ID *)
  SingleID_Cv2 AT D1202 : DWORD;  (* 单机出库ID *)
  Alarm_record : ARRAY [1..48] OF BOOL;  (* Alarm_record *)
  Cv1_Fork_Zero_Pos : BOOL;  (* 入库Fork_在零点 *)
  Cv2_Fork_Zero_Pos : BOOL;  (* 出库Fork_在零点 *)
  CCLink_R : CCLink_R;
  CCLink_W : CCLink_W;
  CCLink_W_Control_Bit : CCLink_W_Control_Bit;
  CCLink_R_Status_Bit : CCLink_R_Status_Bit;
  Start_Rising : BOOL;  (* 启动上升沿 *)
  Initialization_Done : BOOL;  (* 初始化完成 *)
  Device_Initialization : BOOL;  (* 初始化开始 *)
  HMI_Screen AT D5034 : INT;  (* HMI画面切换 *)
  Alarm_Rising : BOOL;  (* 报警上升沿 *)
  Home_Button AT M704 : BOOL;  (* 回原点按钮 *)
  Device_Home AT M705 : BOOL;  (* 回原点中 *)
  Home_Done AT M706 : BOOL;  (* 回原点完成 *)
  SingleAGVPurpose_Cv2 AT D1204 : INT;  (* 单机出库AGV目的 *)
  Stacker_Picking_Goods : BOOL;  (* 堆垛机取货中 *)
  Heartbeat : INT;
  A01_TimeOut AT M707 : BOOL;  (* A01断连 *)
  Q0 : ARRAY [1..2] OF RFID;
  RFID_CV1 : STRING[12];  (* RFID_入 *)
  RFID_CV2 : STRING[12];  (* RFID_出 *)
  Warning_Code AT D1206 : INT;
  AGV_CVArea AT M708 : BOOL;  (* AGV在区域内 *)
END_VAR

// global labels: Drive
VAR_GLOBAL
  Axle_IN_Sew_Read : Sew_Read;
  Axle_OUT_Sew_Read : Sew_Read;
  Axle_IN_Sew_Write : Sew_Write;
  Axle_OUT_Sew_Write : Sew_Write;
  Axle_IN_Sew_Status_Bit : Sew_Status_Bit;
  Axle_OUT_Sew_Status_Bit : Sew_Status_Bit;
  Axle_IN_Sew_Control_Bit : Sew_Control_Bit;
  Axle_OUT_Sew_Control_Bit : Sew_Control_Bit;
  Axle_IN_Status AT D180 : WORD;
  Axle_OUT_Status AT D181 : WORD;
  Axle_IN_Alalm AT D182 : WORD;
  Axle_OUT_Alalm AT D183 : WORD;
  Axle_IN_Pos AT D164 : DINT;
  Axle_OUT_Pos AT D174 : DINT;
  Execute_Pos_CV1 : BOOL;  (* 开始定位_IN *)
  Execute_Pos_CV2 : BOOL;  (* 开始定位_OUT *)
  CV1_Fork_Actual_Position AT D184 : DINT;  (* 入库货叉实际位置 *)
  CV1_Fork_Current_Position AT D186 : DINT;  (* 入库货叉当前位置 *)
  CV2_Fork_Actual_Position AT D188 : DINT;  (* 出库货叉实际位置 *)
  CV2_Fork_Current_Position AT D190 : DINT;  (* 出库货叉当前位置 *)
  CV1_Fork_Actual_Position_1 AT D162 : DINT;  (* 入库货叉实际位置_1 *)
  CV2_Fork_Actual_Position_1 AT D172 : DINT;  (* 出库货叉实际位置_1 *)
  CV1_Fork_Stretch_Enable : BOOL;  (* 入库货叉伸出允许 *)
  CV1_Fork_Back_Enable : BOOL;  (* 入库货叉缩回允许 *)
  CV2_Fork_Stretch_Enable : BOOL;  (* 出库货叉伸出允许 *)
  CV2_Fork_Back_Enable : BOOL;  (* 出库货叉缩回允许 *)
  CV1_Fork_Positioning_Done : BOOL;  (* 入库货叉定位到达 *)
  CV2_Fork_Positioning_Done : BOOL;  (* 出库货叉定位到达 *)
  CV1_Target_Position : DINT;  (* 入库定位位置 *)
  CV2_Target_Position : DINT;  (* 出库定位位置 *)
  AGV_IN_LightCurtain_Invalid : BOOL;  (* AGV入侧光栅屏蔽中 *)
  AGV_Out_LightCurtain_Invalid : BOOL;  (* AGV出侧光栅屏蔽中 *)
END_VAR

PROGRAM MAIN
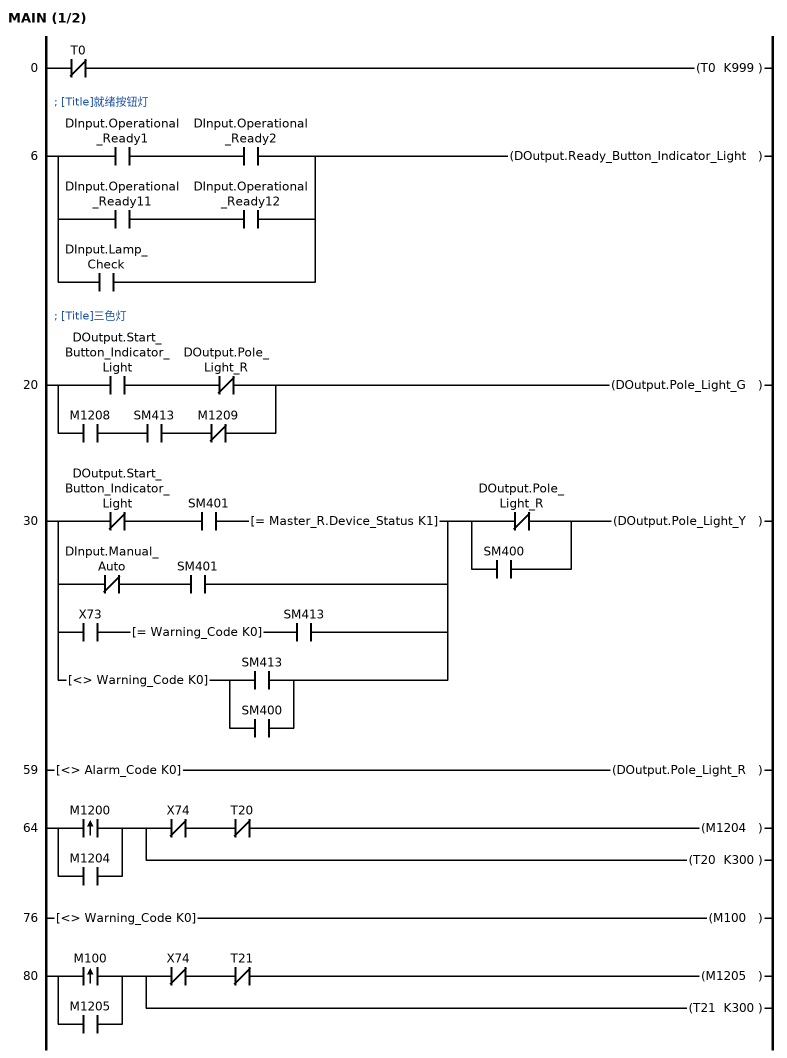
0     LDI     T0
      OUT     T0 K999
; [Title]就绪按钮灯
6     LD      DInput.Operational_Ready1
      AND     DInput.Operational_Ready2
      LD      DInput.Operational_Ready11
      AND     DInput.Operational_Ready12
      ORB
      OR      DInput.Lamp_Check
      OUT     DOutput.Ready_Button_Indicator_Light
; [Title]三色灯
20    LD      DOutput.Start_Button_Indicator_Light
      ANI     DOutput.Pole_Light_R
      LD      M1208
      AND     SM413
      ANI     M1209
      ORB
      OUT     DOutput.Pole_Light_G
30    LDI     DOutput.Start_Button_Indicator_Light
      AND     SM401
      AND=    Master_R.Device_Status K1
      LDI     DInput.Manual_Auto
      AND     SM401
      ORB
      LD      X73
      AND=    Warning_Code K0
      AND     SM413
      ORB
      LD<>    Warning_Code K0
      LD      SM413
      OR      SM400
      ANB
      ORB
      LDI     DOutput.Pole_Light_R
      OR      SM400
      ANB
      OUT     DOutput.Pole_Light_Y
59    LD<>    Alarm_Code K0
      OUT     DOutput.Pole_Light_R
64    LDP     M1200
      OR      M1204
      MPS
      ANI     X74
      ANI     T20
      OUT     M1204
      MPP
      OUT     T20 K300
76    LD<>    Warning_Code K0
      OUT     M100
80    LDP     M100
      OR      M1205
      MPS
      ANI     X74
      ANI     T21
      OUT     M1205
      MPP
      OUT     T21 K300
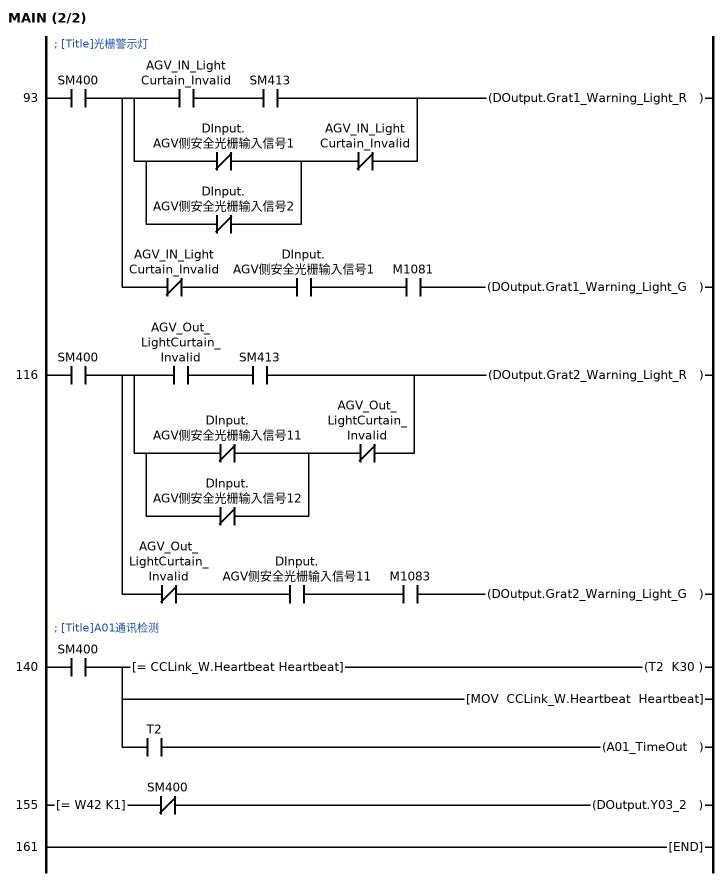
; [Title]光栅警示灯
93    LD      SM400
      MPS
      LD      AGV_IN_LightCurtain_Invalid
      AND     SM413
      LDI     DInput.AGV侧安全光栅输入信号1
      ORI     DInput.AGV侧安全光栅输入信号2
      ANI     AGV_IN_LightCurtain_Invalid
      ORB
      ANB
      OUT     DOutput.Grat1_Warning_Light_R
      MPP
      ANI     AGV_IN_LightCurtain_Invalid
      AND     DInput.AGV侧安全光栅输入信号1
      AND     M1081
      OUT     DOutput.Grat1_Warning_Light_G
116   LD      SM400
      MPS
      LD      AGV_Out_LightCurtain_Invalid
      AND     SM413
      LDI     DInput.AGV侧安全光栅输入信号11
      ORI     DInput.AGV侧安全光栅输入信号12
      ANI     AGV_Out_LightCurtain_Invalid
      ORB
      ANB
      OUT     DOutput.Grat2_Warning_Light_R
      MPP
      ANI     AGV_Out_LightCurtain_Invalid
      AND     DInput.AGV侧安全光栅输入信号11
      AND     M1083
      OUT     DOutput.Grat2_Warning_Light_G
; [Title]A01通讯检测
140   LD      SM400
      MPS
      AND=    CCLink_W.Heartbeat Heartbeat
      OUT     T2 K30
      MPP
      MOV     CCLink_W.Heartbeat Heartbeat
      AND     T2
      OUT     A01_TimeOut
155   LD=     W42 K1
      ANI     SM400
      OUT     DOutput.Y03_2
161   END
END_PROGRAM

PROGRAM IO
(*输入*)
DInput.In_Power:=X60;
DInput.X01_1:=X61;
DInput.B01_Emergency_Stop_Circuit1:=X62;
DInput.B01_Emergency_Stop_Circuit2:=X63;
DInput.B01_Grating_Circuit1:=X64;
DInput.B01_Grating_Circuit2:=X65;
DInput.B01_Safety_Door_Circuit1:=X66;
DInput.B01_Safety_Door_Circuit2:=X67;
DInput.AO1Safety_Circuit1:=X68;
DInput.AO1Safety_Circuit2:=X69;
DInput.B02_Emergency_Stop_Circuit1:=X6A;
DInput.B02_Emergency_Stop_Circuit2:=X6B;
DInput.B02_Grating_Circuit1:=X6C;
DInput.B02_Grating_Circuit2:=X6D;
DInput.B02_Safety_Door_Circuit1:=X6E;
DInput.B02_Safety_Door_Circuit2:=X6F;

DInput.Manual_Auto:=X70;
DInput.Single_OnLine:=X71;
DInput.X02_2:=X72;
DInput.Admin:=X73;
DInput.Alarm_Reset:=X74;
DInput.Ready_Button:=X75;
DInput.Start_Button:=X76;
DInput.Pause_Button:=X77;
DInput.Lamp_Check:=X78;
DInput.X09_2:=X79;
DInput.Operational_Ready1:=X7A;
DInput.Operational_Ready2:=X7B;
DInput.Operational_Ready11:=X7C;
DInput.Operational_Ready12:=X7D;
DInput.Air_Error:=X7E;
DInput.X0F_2:=X7F;

DInput.CV01顶升上限检测:=X80;
DInput.CV01顶升下限检测:=X81;
DInput.CV01顶升故障检测:=X82;
DInput.CV01顶升电源检测:=X83;
DInput.CV01物料停止检测:=X84;
DInput.X05_3:=X85;
DInput.CV01伸缩中位检测1:=X86;
DInput.CV01伸缩中位检测2:=X87;
DInput.CV01伸缩极限检测:=NOT X88;
DInput.CV01伸缩电源检测:=X89;
DInput.CV01AGV物料检测:=X8A;
DInput.CV01AGV本体检测1:=X8B;
DInput.CV01AGV本体检测2:=X8C;
DInput.CV01超宽检测1:=X8D;
DInput.CV01超宽检测2:=X8E;
DInput.CV01超高检测:=X8F;

DInput.Bx03顶升上限检测:=X90;
DInput.Bx03顶升下限检测:=X91;
DInput.Bx03顶升故障检测:=X92;
DInput.Bx03顶升电源检测:=X93;
DInput.Bx03物料停止检测:=X94;
DInput.Bx03物料减速检测:=X95;
DInput.CV02伸缩中位检测1:=X96;
DInput.CV02伸缩中位检测2:=X97;
DInput.CV02伸缩极限检测:=NOT X98;
DInput.Bx03伸缩电源检测:=X99;
DInput.Bx03AGV物料检测:=X9A;
DInput.Bx03AGV本体检测1:=X9B;
DInput.Bx03AGV本体检测2:=X9C;
DInput.X0D_4:=X9D;
DInput.X0E_4:=X9E;
DInput.X0F_4:=X9F;

DInput.Bx02顶升上限检测:=XA0;
DInput.Bx02顶升下限检测:=XA1;
DInput.Bx02顶升故障检测:=XA2;
DInput.Bx02顶升电源检测:=XA3;
DInput.Bx02物料到位检测:=XA4;
DInput.Bx02物料减速检测:=XA5;
DInput.Bx02输送故障检测:=XA6;
DInput.Bx02输送电源检测:=XA7;
DInput.Bx04顶升上限检测:=XA8;
DInput.Bx04顶升下限检测:=XA9;
DInput.Bx04顶升故障检测:=XAA;
DInput.Bx04顶升电源检测:=XAB;
DInput.Bx04物料到位检测:=XAC;
DInput.X0D_5:=XAD;
DInput.Bx04输送故障检测:=XAE;
DInput.Bx04输送电源检测:=XAF;

DInput.AGV侧安全光栅输入信号1:=XB0;
DInput.AGV侧安全光栅输入信号2:=XB1;
DInput.AGV侧安全光栅输入信号11:=XB2;
DInput.AGV侧安全光栅输入信号12:=XB3;
DInput.CV_IN侧安全光栅输入信号1:=XB4;
DInput.CV_IN侧安全光栅输入信号2:=XB5;
DInput.CV_Out侧安全光栅输入信号1:=XB6;
DInput.CV_Out侧安全光栅输入信号2:=XB7;
DInput.X08_6:=XB8;
DInput.X09_6:=XB9;
DInput.安全门1输入信号1:=XBA;
DInput.安全门1输入信号2:=XBB;
DInput.解锁1安全门:=XBC;
DInput.X0D_6:=XBD;
DInput.X0E_6:=XBE;
DInput.X0F_6:=XBF;

IF W42=1 THEN 
DInput.Photonic1_output1:=XC0;
DInput.Photonic1_output2:=XC1;
DInput.Photonic1_output3:=XC2;
DInput.Photonic1_output4:=XC3;
DInput.Photonic1_Go:=XC4;
ELSIF W42=2 THEN 
DInput.Photonic4_output1:=XC0;
DInput.Photonic4_output2:=XC1;
DInput.Photonic4_output3:=XC2;
DInput.Photonic4_output4:=XC3;
DInput.Photonic4_Go:=XC4;
END_IF;	
DInput.X05_7:=XC5;
DInput.Photonic2_output1:=XC6;
DInput.Photonic2_output2:=XC7;
DInput.Photonic2_output3:=XC8;
DInput.Photonic2_output4:=XC9;
DInput.Photonic2_Go:=XCA;
DInput.X0B_7:=XCB;
DInput.Photonic3_output1:=XCC;
DInput.Photonic3_output2:=XCD;
DInput.Photonic3_output3:=XCE;
DInput.Photonic3_output4:=XCF;

DInput.Photonic3_Go:=XD0;
DInput.X01_8:=XD1;
IF W42=1 THEN 
DInput.Photonic4_output1:=XD2;
DInput.Photonic4_output2:=XD3;
DInput.Photonic4_output3:=XD4;
DInput.Photonic4_output4:=XD5;
DInput.Photonic4_Go:=XD6;
ELSIF W42=2 THEN 
DInput.Photonic1_output1:=XD2;
DInput.Photonic1_output2:=XD3;
DInput.Photonic1_output3:=XD4;
DInput.Photonic1_output4:=XD5;
DInput.Photonic1_Go:=XD6;
END_IF;	
DInput.X07_8:=XD7;
DInput.X08_8:=XD8;
DInput.X09_8:=XD9;
DInput.X0A_8:=XDA;
DInput.X0B_8:=XDB;
DInput.X0C_8:=XDC;
DInput.X0D_8:=XDD;
DInput.X0E_8:=XDE;
DInput.X0F_8:=XDF;

(*输出*)
YE0:=DOutput.Pole_Light_R OR DInput.Lamp_Check;
YE1:=DOutput.Pole_Light_Y OR DInput.Lamp_Check;
YE2:=DOutput.Pole_Light_G OR DInput.Lamp_Check;
YE3:=DOutput.HA01_Sound1;
YE4:=DOutput.HA01_Sound2;
YE5:=DOutput.HA01_Sound3;
YE6:=DOutput.HA01_Sound4;
YE7:=DOutput.Y07_1;
YE8:=DOutput.Ready_Button_Indicator_Light OR DInput.Lamp_Check;
YE9:=DOutput.Start_Button_Indicator_Light OR DInput.Lamp_Check;
YEA:=DOutput.Pause_Button_Indicator_Light OR DInput.Lamp_Check;
YEB:=DOutput.Y0B_1;
YEC:=DOutput.Y0C_1;
YED:=DOutput.Y0D_1;
YEE:=DOutput.SafetyDoor_Indicator_Light;
YEF:=DOutput.Unlock_SafetyDoor;

YF0:=DOutput.CV1_JackingUP_Fork_Run;
YF1:=DOutput.CV1_JackingDown_Fork_Run;
YF2:=DOutput.CV1_Jacking_Fork_Reset;
YF3:=DOutput.Y03_2;
YF4:=DOutput.Grat1_Warning_Light_R OR DInput.Lamp_Check;
YF5:=DOutput.Grat1_Warning_Light_G OR DInput.Lamp_Check;
YF6:=DOutput.CV1_JackingUP_Run;
YF7:=DOutput.CV1_JackingDown_Run;
YF8:=DOutput.CV1_Jacking_Reset;
YF9:=DOutput.Y09_2;
YFA:=DOutput.CV1_ConveyingIN_Run;
YFB:=DOutput.CV1_ConveyingOut_Run;
YFC:=DOutput.CV1_Conveying_SpeedA;
YFD:=DOutput.CV1_Conveying_SpeedB;
YFE:=DOutput.CV1_Conveying_Reset;
YFF:=DOutput.Y0F_2;

Y100:=DOutput.CV2_JackingUP_Fork_Run;
Y101:=DOutput.CV2_JackingDown_Fork_Run;
Y102:=DOutput.CV2_Jacking_Fork_Reset;
Y103:=DOutput.Y03_3;
Y104:=DOutput.Grat2_Warning_Light_R OR DInput.Lamp_Check;
Y105:=DOutput.Grat2_Warning_Light_G OR DInput.Lamp_Check;
Y106:=DOutput.CV2_JackingUP_Run;
Y107:=DOutput.CV2_JackingDown_Run;
Y108:=DOutput.CV2_Jacking_Reset;
Y109:=DOutput.Y09_3;
Y10A:=DOutput.CV2_ConveyingIN_Run;
Y10B:=DOutput.CV2_ConveyingOut_Run;
Y10C:=DOutput.CV2_Conveying_SpeedA;
Y10D:=DOutput.CV2_Conveying_SpeedB;
Y10E:=DOutput.CV2_Conveying_Reset;
Y10F:=DOutput.Y0F_3;

IF W42=1 THEN 
Y110:=DOutput.Photonic1_Input1;
Y111:=DOutput.Photonic1_Input2;
Y112:=DOutput.Photonic1_Input3;
Y113:=DOutput.Photonic1_Input4;
ELSIF W42=2 THEN 
Y110:=DOutput.Photonic4_Input1;
Y111:=DOutput.Photonic4_Input2;
Y112:=DOutput.Photonic4_Input3;
Y113:=DOutput.Photonic4_Input4;
END_IF;	
Y114:=DOutput.Photonic2_Input1;
Y115:=DOutput.Photonic2_Input2;
Y116:=DOutput.Photonic2_Input3;
Y117:=DOutput.Photonic2_Input4;
Y118:=DOutput.Photonic3_Input1;
Y119:=DOutput.Photonic3_Input2;
Y11A:=DOutput.Photonic3_Input3;
Y11B:=DOutput.Photonic3_Input4;
IF W42=1 THEN 
Y11C:=DOutput.Photonic4_Input1;
Y11D:=DOutput.Photonic4_Input2;
Y11E:=DOutput.Photonic4_Input3;
Y11F:=DOutput.Photonic4_Input4;
ELSIF W42=2 THEN 
Y11C:=DOutput.Photonic1_Input1;
Y11D:=DOutput.Photonic1_Input2;
Y11E:=DOutput.Photonic1_Input3;
Y11F:=DOutput.Photonic1_Input4;	
END_IF;	
	
Y120:=DOutput.Y00_5;
Y121:=DOutput.Y01_5;
Y122:=DOutput.Y02_5;
Y123:=DOutput.Y03_5;
Y124:=DOutput.Y04_5;
Y125:=DOutput.Y05_5;
Y126:=DOutput.Invalid_CV_IN_Grat1;
Y127:=DOutput.Invalid_CV_IN_Grat2;
Y128:=DOutput.Y08_5;
Y129:=DOutput.Invalid_CV_OUT_Grat1;
Y12A:=DOutput.Invalid_CV_OUT_Grat2;
Y12B:=DOutput.Y0B_5;
Y12C:=DOutput.Invalid_SafetyDoor1;
Y12D:=DOutput.Invalid_SafetyDoor2;
Y12E:=DOutput.Y0E_5;
Y12F:=DOutput.Y0F_5;

Deliver_In.入库口顶升上限检测:=DInput.Bx02顶升上限检测;
Deliver_In.入库口顶升下限检测:=DInput.Bx02顶升下限检测;
Deliver_In.货叉顶升上限检测:=DInput.CV01顶升上限检测;
Deliver_In.货叉顶升下限检测:=DInput.CV01顶升下限检测;
Deliver_In.入库口物料检测:=TS10;
 OUT_T(DInput.Bx02物料到位检测,TC10,20);
Deliver_In.入库口减速检测:=DInput.Bx02物料减速检测;
Deliver_In.货叉位置物料检测:=DInput.CV01物料停止检测;
Deliver_In.货叉伸出到位:=CV1_Fork_Positioning_Done AND Deliver_In.货叉伸出控制;
Deliver_In.货叉缩回到位:=DInput.CV01伸缩中位检测1 AND DInput.CV01伸缩中位检测2 AND Execute_Pos_CV1=FALSE ;


Deliver_OUT.出库口顶升上限检测:=DInput.Bx04顶升上限检测;
Deliver_OUT.出库口顶升下限检测:=DInput.Bx04顶升下限检测;
Deliver_OUT.货叉顶升上限检测:=DInput.Bx03顶升上限检测;
Deliver_OUT.货叉顶升下限检测:=DInput.Bx03顶升下限检测;
Deliver_OUT.出库口物料检测:=DInput.Bx04物料到位检测;
Deliver_OUT.货叉位置减速检测:=DInput.Bx03物料减速检测;
Deliver_OUT.货叉位置物料检测:=TS11;
 OUT_T(DInput.Bx03物料停止检测,TC11,20);
Deliver_OUT.货叉伸出到位:=CV2_Fork_Positioning_Done AND Deliver_OUT.货叉伸出控制;
Deliver_OUT.货叉缩回到位:=DInput.CV02伸缩中位检测1 AND DInput.CV02伸缩中位检测2  AND Execute_Pos_CV2=FALSE ;
END_PROGRAM

PROGRAM Func
VAR
  Store_1 : Store;
  Outbound_1 : Outbound;
END_VAR
(*急停*)
E_Stop:=DInput.B01_Emergency_Stop_Circuit1 AND DInput.B01_Emergency_Stop_Circuit2;
IF E_Stop=FALSE OR Alarm_Code<>0 OR mode=2 OR DOutput.Ready_Button_Indicator_Light=FALSE THEN
    DOutput.Start_Button_Indicator_Light:=FALSE;
    DOutput.Pause_Button_Indicator_Light:=FALSE;
    Device_Initialization:=FALSE;
END_IF;

(*启动按钮*)
IF DInput.Start_Button AND mode<=1  AND DOutput.Ready_Button_Indicator_Light AND Alarm_Code=0  AND DOutput.Pause_Button_Indicator_Light=FALSE THEN
	DOutput.Start_Button_Indicator_Light:=TRUE;
END_IF;
(*暂停按钮*)
IF DInput.Pause_Button AND DOutput.Start_Button_Indicator_Light THEN
	DOutput.Pause_Button_Indicator_Light:=TRUE;
	DOutput.Start_Button_Indicator_Light:=FALSE;
ELSIF 
	Device_Station THEN
	DOutput.Pause_Button_Indicator_Light:=FALSE;
END_IF;
 
 (*AGV光栅屏蔽*)
 IF HMI.Invalid_AGV_IN_Grat OR Deliver_In.AGV进入中 OR (W42=2 AND Deliver_Out.AGVl离开中 )THEN
 	AGV_IN_LightCurtain_Invalid:=TRUE;
 ELSE
 	AGV_IN_LightCurtain_Invalid:=FALSE;
 END_IF;
  IF HMI.Invalid_AGV_OUT_Grat OR Deliver_Out.AGVl离开中 THEN
 	AGV_Out_LightCurtain_Invalid:=TRUE;
 ELSE
 	AGV_Out_LightCurtain_Invalid:=FALSE;
  END_IF;
  
 IF DInput.CV01伸缩中位检测2=FALSE OR HMI.Invalid_CV_IN_Grat OR Axle_IN_Sew_Control_Bit.Ramp_Bus_StartStop=TRUE THEN
 	DOutput.Invalid_CV_IN_Grat1:=TRUE;
 	DOutput.Invalid_CV_IN_Grat2:=TRUE;
 ELSE
 	DOutput.Invalid_CV_IN_Grat1:=FALSE;
 	DOutput.Invalid_CV_IN_Grat2:=FALSE;
 END_IF;
 IF  DInput.CV02伸缩中位检测2=FALSE OR HMI.Invalid_CV_OUT_Grat OR Axle_Out_Sew_Control_Bit.Ramp_Bus_StartStop=TRUE THEN
 	DOutput.Invalid_CV_OUT_Grat1 :=TRUE;
 	DOutput.Invalid_CV_OUT_Grat2 :=TRUE;
 ELSE
 	DOutput.Invalid_CV_OUT_Grat1 :=FALSE;
 	DOutput.Invalid_CV_OUT_Grat2 :=FALSE;
 END_IF;
  IF HMI.Invalid_SafetyDoor THEN
 	DOutput.Invalid_SafetyDoor1  :=TRUE;
 	DOutput.Invalid_SafetyDoor2  :=TRUE;
 ELSE
 	DOutput.Invalid_SafetyDoor1  :=FALSE;
 	DOutput.Invalid_SafetyDoor2  :=FALSE;
 END_IF;
 
  (*解锁1安全门 *)
 IF DInput.解锁1安全门 THEN
 	DOutput.SafetyDoor_Indicator_Light:=FALSE;
 	DOutput.Unlock_SafetyDoor:=TRUE;
 ELSE
 	DOutput.SafetyDoor_Indicator_Light:=TRUE;
 	DOutput.Unlock_SafetyDoor:=FALSE;
 END_IF;
 
 (*SM411~SM414‌：分别10ms、100ms、1s、1min的时钟脉冲信号*)
(*设备静止中*)
IF Deliver_In.Step1=0 AND Deliver_Out.Step1=0 THEN
	Device_Station :=TRUE;
ELSE
	Device_Station :=FALSE;
END_IF;

 (*模式*)
 IF DInput.Manual_Auto=FALSE THEN
  	mode :=2;
 ELSE
  	IF DInput.Single_OnLine=FALSE THEN
  		mode :=1;
  	ELSE
  		mode :=0;
  	END_IF;
 END_IF;
  
(*模式显示*)
OnLine_Mode:=Mode=0;
Single_Mode:=Mode=1;
Manual_Mode:=Mode=2;

(*语言切换*)
IF Language>3 OR Language=0 THEN
	Language:=1;
END_IF;
INCP(Language_Switch,Language);

(*密码权限-管理者*)
IF DInput.Admin=FALSE THEN
	Password:=0;
	DOutput.HA01_Sound4:=FALSE;
	HMI.Invalid_CV_IN_Grat:=FALSE;
	HMI.Invalid_CV_OUT_Grat:=FALSE;
	HMI.Invalid_SafetyDoor:=FALSE;
ELSE
	(*DOutput.HA01_Sound4:=TRUE;*)
	DOutput.HA01_Sound4:=FALSE;
END_IF;
 	
 (*自动流程入库*)
Store_1();
 
 (*自动流程出库*)
Outbound_1();
 
  (*Fork_在零点*)
Cv1_Fork_Zero_Pos:=DInput.CV01伸缩中位检测1 AND DInput.CV01伸缩中位检测2 AND ABS(CV1_Fork_Current_Position)<=5 ;
Cv2_Fork_Zero_Pos:=DInput.CV02伸缩中位检测1  AND DInput.CV02伸缩中位检测2  AND ABS(CV2_Fork_Current_Position)<=5 ;
 
 (*手动允许*)
 IF CV1_Fork_Current_Position<=parameter.CV1_Fork_Position_Set AND DInput.CV01伸缩极限检测=FALSE AND DOutput.Ready_Button_Indicator_Light THEN
 	CV1_Fork_Stretch_Enable:=TRUE;
 ELSE
 	CV1_Fork_Stretch_Enable:=FALSE;
 END_IF;
  IF CV1_Fork_Current_Position>-1  AND DOutput.Ready_Button_Indicator_Light THEN
 	CV1_Fork_Back_Enable:=TRUE;
 ELSE
 		CV1_Fork_Back_Enable:=FALSE;
  END_IF;
  
  IF CV2_Fork_Current_Position<=parameter.CV2_Fork_Position_Set AND DInput.CV02伸缩极限检测=FALSE  AND DOutput.Ready_Button_Indicator_Light THEN
 	  CV2_Fork_Stretch_Enable:=TRUE;
 ELSE
 	  CV2_Fork_Stretch_Enable:=FALSE;
 END_IF;
  IF CV2_Fork_Current_Position>-1  AND DOutput.Ready_Button_Indicator_Light THEN
 	    CV2_Fork_Back_Enable:=TRUE;
 ELSE
 		CV2_Fork_Back_Enable:=FALSE;
  END_IF;
  
   (*手动模式*)
IF Mode=2 THEN
	    Axle_IN_Sew_Control_Bit.Forward_Jog:=Manual.手动入库货叉伸出 AND CV1_Fork_Stretch_Enable ;
		Axle_IN_Sew_Control_Bit.Reverse_Jog:=Manual.手动入库货叉缩回 AND CV1_Fork_Back_Enable;
		Axle_OUT_Sew_Control_Bit.Forward_Jog:=Manual.手动出库货叉伸出 AND CV2_Fork_Stretch_Enable;
		Axle_OUT_Sew_Control_Bit.Reverse_Jog:=Manual.手动出库货叉缩回 AND CV2_Fork_Back_Enable;
		
		IF Axle_IN_Sew_Control_Bit.Forward_Jog OR Axle_IN_Sew_Control_Bit.Reverse_Jog THEN
			Axle_IN_Sew_Write.Set_Mode:=100;
			Axle_IN_Sew_Control_Bit.Enable_Emergency_Stop:=TRUE;
			Axle_IN_Sew_Control_Bit.Enable_Application_Stop:=TRUE;
			Axle_IN_Sew_Write.Rated_Speed:=100;
		END_IF;
		
		IF Axle_OUT_Sew_Control_Bit.Forward_Jog OR Axle_OUT_Sew_Control_Bit.Reverse_Jog THEN
			Axle_OUT_Sew_Write.Set_Mode:=100;
			Axle_OUT_Sew_Control_Bit.Enable_Emergency_Stop:=TRUE;
			Axle_OUT_Sew_Control_Bit.Enable_Application_Stop:=TRUE;
			Axle_OUT_Sew_Write.Rated_Speed:=100;
		END_IF;
END_IF;

 (*自动模式*)
 (*入库*)
IF( Deliver_In.货叉伸出控制  OR (Manual.自动入库货叉伸出 AND Manual_Mode)) AND DOutput.Ready_Button_Indicator_Light  THEN
	CV1_Target_Position:=(parameter.CV1_Fork_Position_Set+parameter.CV1_Fork_Pos_Offset);
	Axle_IN_Pos:=CV1_Target_Position*10;
	Execute_Pos_CV1:=TRUE;
END_IF;
IF( Deliver_In.货叉缩回控制 OR (Manual.自动入库货叉缩回 AND Manual_Mode))AND DOutput.Ready_Button_Indicator_Light THEN 
	CV1_Target_Position:=0;
		Axle_IN_Pos:=CV1_Target_Position;
		Execute_Pos_CV1:=TRUE;
END_IF;
IF Execute_Pos_CV1  THEN
	        Axle_IN_Sew_Write.Set_Mode:=400;
			Axle_IN_Sew_Control_Bit.Enable_Emergency_Stop:=TRUE;
			Axle_IN_Sew_Control_Bit.Enable_Application_Stop:=TRUE;
			Axle_IN_Sew_Control_Bit.Ramp_Bus_StartStop:=TRUE;
			Axle_IN_Sew_Write.Rated_Speed:=parameter.CV1_Fork_Speed_Set;
END_IF;

(*出库*)
   IF( Deliver_OUT.货叉伸出控制  OR (Manual.自动出库货叉伸出  AND Manual_Mode)) AND DOutput.Ready_Button_Indicator_Light  THEN
	  CV2_Target_Position:=(parameter.CV2_Fork_Position_Set+parameter.CV2_Fork_Pos_Offset);
	  Axle_OUT_Pos:=CV2_Target_Position*10;
	  Execute_Pos_CV2:=TRUE;
	END_IF;
	IF (Deliver_OUT.货叉缩回控制 OR (Manual.自动出库货叉缩回 AND Manual_Mode)) AND DOutput.Ready_Button_Indicator_Light  THEN
		CV2_Target_Position:=0;
		Axle_OUT_Pos:=CV2_Target_Position;
		Execute_Pos_CV2:=TRUE;
	END_IF;
	IF Execute_Pos_CV2 THEN 
	       Axle_OUT_Sew_Write.Set_Mode:=400;
			Axle_OUT_Sew_Control_Bit.Enable_Emergency_Stop:=TRUE;
			Axle_OUT_Sew_Control_Bit.Enable_Application_Stop:=TRUE;
			Axle_OUT_Sew_Control_Bit.Ramp_Bus_StartStop:=TRUE;
			Axle_OUT_Sew_Write.Rated_Speed:=parameter.CV2_Fork_Speed_Set;	
END_IF;

(*加减速度*)
Axle_IN_Sew_Write.Acceleration:=parameter.CV1_Fork_Acceleration_Set;
Axle_IN_Sew_Write.Deceleration:=parameter.CV1_Fork_Deceleration_Set;
Axle_OUT_Sew_Write.Acceleration:=parameter.CV2_Fork_Acceleration_Set;
Axle_OUT_Sew_Write.Deceleration:=parameter.CV2_Fork_Deceleration_Set;

(*定位到达*)
IF ABS(CV1_Fork_Current_Position-CV1_Target_Position)<20 THEN
      CV1_Fork_Positioning_Done:=TRUE;
ELSE
	CV1_Fork_Positioning_Done:=FALSE;
END_IF;
IF ABS(CV2_Fork_Current_Position-CV2_Target_Position)<20 THEN
      CV2_Fork_Positioning_Done:=TRUE;
ELSE
	CV2_Fork_Positioning_Done:=FALSE;
END_IF;

IF Axle_IN_Sew_Status_Bit.Position_Arrive AND Axle_IN_Sew_Control_Bit.Ramp_Bus_StartStop  AND CV1_Fork_Positioning_Done THEN
	Execute_Pos_CV1:=FALSE;
END_IF;
IF Axle_OUT_Sew_Status_Bit.Position_Arrive AND Axle_OUT_Sew_Control_Bit.Ramp_Bus_StartStop  AND CV2_Fork_Positioning_Done THEN
	Execute_Pos_CV2:=FALSE;
END_IF;

(*复位*)
IF Axle_IN_Sew_Control_Bit.Forward_Jog=FALSE  AND Axle_IN_Sew_Control_Bit.Reverse_Jog=FALSE  AND Execute_Pos_CV1=FALSE THEN
	Axle_IN_Sew_Control_Bit.Enable_Emergency_Stop:=FALSE;
	Axle_IN_Sew_Control_Bit.Enable_Application_Stop:=FALSE;
	Axle_IN_Sew_Control_Bit.Ramp_Bus_StartStop:=FALSE;
END_IF;

IF Axle_OUT_Sew_Control_Bit.Forward_Jog=FALSE  AND Axle_OUT_Sew_Control_Bit.Reverse_Jog=FALSE  AND Execute_Pos_CV2=FALSE THEN
	Axle_OUT_Sew_Control_Bit.Enable_Emergency_Stop:=FALSE;
	Axle_OUT_Sew_Control_Bit.Enable_Application_Stop:=FALSE;
	Axle_OUT_Sew_Control_Bit.Ramp_Bus_StartStop:=FALSE;
END_IF;

(*货叉当前位置换算*)
CV1_Fork_Actual_Position:=CV1_Fork_Actual_Position_1/10;
CV1_Fork_Current_Position:=CV1_Fork_Actual_Position-parameter.CV1_Fork_Pos_Offset;

CV2_Fork_Actual_Position:=CV2_Fork_Actual_Position_1/10;
CV2_Fork_Current_Position:=CV2_Fork_Actual_Position-parameter.CV2_Fork_Pos_Offset;

(*故障及状态获取*)
IF  Axle_IN_Sew_Status_Bit.Error THEN
	Axle_IN_Alalm := Axle_IN_Sew_Read.Main_Status_Fault;
	Axle_IN_Status := 0;
ELSE
	Axle_IN_Alalm:=0 ;
	Axle_IN_Status:=Axle_IN_Sew_Read.Main_Status_Fault ;
END_IF;
IF  Axle_OUT_Sew_Status_Bit.Error THEN
	Axle_OUT_Alalm:=Axle_OUT_Sew_Read.Main_Status_Fault;
	Axle_OUT_Status:=0;
ELSE
	Axle_OUT_Alalm:=0;
	Axle_OUT_Status:=Axle_OUT_Sew_Read.Main_Status_Fault;
END_IF;

(*急停*)
IF E_Stop=FALSE OR Alarm_Code<>0 THEN
	Execute_Pos_CV1:=FALSE;
	Execute_Pos_CV2:=FALSE;
	Axle_IN_Sew_Control_Bit.Enable_Emergency_Stop:=FALSE;
	Axle_IN_Sew_Control_Bit.Enable_Application_Stop:=FALSE;
	Axle_IN_Sew_Control_Bit.Ramp_Bus_StartStop:=FALSE;
	Axle_OUT_Sew_Control_Bit.Enable_Emergency_Stop:=FALSE;
	Axle_OUT_Sew_Control_Bit.Enable_Application_Stop:=FALSE;
	Axle_OUT_Sew_Control_Bit.Ramp_Bus_StartStop:=FALSE;
END_IF;

(*设备状态*)
Master_R.Device_Status:=0;
IF Mode<=1 AND Alarm_Code=0 AND DOutput.Start_Button_Indicator_Light AND Initialization_Done THEN 
	Master_R.Device_Status:=1;
END_IF;
IF Alarm_Code<>0 THEN 
	Master_R.Device_Status:=3;
END_IF;

(*回原点*)
IF Home_Button AND Mode=2 THEN
	Device_Home:=TRUE;
END_IF;
IF Device_Home THEN
	IF Cv1_Fork_Zero_Pos=FALSE  THEN
		Manual.自动入库货叉缩回:=TRUE;
	END_IF;
	IF Cv2_Fork_Zero_Pos=FALSE THEN
		Manual.自动出库货叉缩回:=TRUE;
	END_IF;
	IF  Deliver_In. 入库口顶升下限检测 AND Deliver_In. 货叉顶升下限检测 AND 
		 Deliver_Out.出库口顶升下限检测 AND Deliver_Out.货叉顶升下限检测 AND 
		 Cv1_Fork_Zero_Pos AND Cv2_Fork_Zero_Pos THEN
		 Deliver_In.货叉缩回控制:=FALSE;
		 Deliver_Out.货叉缩回控制:=FALSE;
		 Device_Home:=FALSE;
	END_IF;
END_IF;
IF  Mode<>2 OR Alarm_Code<>0  THEN
	Deliver_In.货叉缩回控制:=FALSE;
	Deliver_Out.货叉缩回控制:=FALSE;
	Device_Home:=FALSE;
END_IF;
 	
(*RFID*)                                    
(*托盘编号信息，最长12位数    RFID字符串长度12*)
IF M340 THEN
	RFID_CV1:='' ;
END_IF;	
IF M341 THEN
	RFID_CV2:='' ;
END_IF;	
IF Deliver_In. 货叉位置物料检测 AND Deliver_In. 货叉顶升下限检测 AND Deliver_In.Step1=0 AND M340=FALSE THEN
    Master_R.CV1_Current_RFID:=RFID_CV1;
END_IF;
IF Deliver_In. 货叉位置物料检测=FALSE AND Deliver_In.入库口物料检测=FALSE  AND Deliver_In.Step1=0 THEN
	Master_R.CV1_Current_RFID:='' ;
END_IF;

IF Deliver_Out. 货叉位置物料检测 AND Deliver_Out. 货叉顶升下限检测  AND Deliver_Out.Step1=0 AND M341=FALSE THEN
    Master_R.CV2_Current_RFID:=RFID_CV2;
END_IF;
IF Deliver_Out. 货叉位置物料检测=FALSE  AND Deliver_Out.Step1=0 THEN
	Master_R.CV2_Current_RFID:='' ;
END_IF;
END_PROGRAM

PROGRAM Alarm
(*IF DInput.输入电源=FALSE AND Alarm_Code=0 THEN
	Alarm_Code:=1;
END_IF;*)

IF DInput.Air_Error AND Alarm_Code=0 THEN
	Alarm_Code:=2;
END_IF;

(*IF E_Stop=FALSE AND Alarm_Code=0 THEN*)
IF E_Stop=FALSE  THEN
	Alarm_Code:=3;
END_IF;

IF Axle_IN_Sew_Status_Bit.Error AND Alarm_Code=0 THEN
	Alarm_Code:=4;
END_IF;
	
IF Axle_OUT_Sew_Status_Bit.Error AND Alarm_Code=0 THEN
	Alarm_Code:=5;
END_IF;
	
(*1：计划不满足，2：RFID不匹配，3：计划不满足，且RFID不匹配。6789*)

(*货叉变频器通讯故障*)	
IF M320 AND Alarm_Code=0 THEN
	Alarm_Code:=10;
END_IF;
IF M322 AND Alarm_Code=0 THEN
	Alarm_Code:=11;
END_IF;
	
(*入库侧*)
IF( DInput.CV01超宽检测1 OR DInput.CV01超宽检测2) AND Alarm_Code=0 AND Mode<>2 THEN
	Alarm_Code:=12;
END_IF;
	
IF DInput.CV01超高检测 AND Alarm_Code=0 AND Mode<>2 THEN
	Alarm_Code:=13;
END_IF;

(*光栅*)	
IF (DInput.AGV侧安全光栅输入信号1=FALSE  OR DInput.AGV侧安全光栅输入信号2=FALSE ) AND AGV_IN_LightCurtain_Invalid =FALSE AND Alarm_Code=0 THEN
	Alarm_Code:=14;
END_IF;
IF( DInput.AGV侧安全光栅输入信号11=FALSE  OR DInput.AGV侧安全光栅输入信号12=FALSE  ) AND AGV_Out_LightCurtain_Invalid =FALSE AND Alarm_Code=0 THEN
	Alarm_Code:=15;
END_IF;
IF( (DInput.CV_IN侧安全光栅输入信号1 =FALSE OR DInput.CV_IN侧安全光栅输入信号2=FALSE)  AND  HMI.Invalid_CV_IN_Grat=FALSE ) AND DInput.CV01伸缩中位检测2 AND Alarm_Code=0 THEN
	Alarm_Code:=16;
END_IF;
IF ((DInput.CV_Out侧安全光栅输入信号1=FALSE  OR DInput.CV_Out侧安全光栅输入信号2=FALSE  )  AND  HMI.Invalid_CV_OUT_Grat=FALSE) AND DInput.CV02伸缩中位检测2 AND  Alarm_Code=0 THEN
	Alarm_Code:=17;
END_IF;
	
(*安全门*)
IF ((DInput.安全门1输入信号1=FALSE   OR DInput.安全门1输入信号2 =FALSE ) AND  HMI.Invalid_SafetyDoor=FALSE)  AND Alarm_Code=0 THEN
	Alarm_Code:=18;
END_IF;

(*入库侧坍塌报警*)
IF CCLink_R_Status_Bit.入库坍塌检测 AND DInput.CV01伸缩中位检测2 AND Alarm_Code=0 AND Mode<>2 THEN
	Alarm_Code:=19;
END_IF;

(*入库口顶升变频器电机故障*)
IF DInput.Bx02输送故障检测 AND   Alarm_Code=0 THEN
	Alarm_Code:=20;
END_IF;

(*入库货叉顶升变频器电机故障*)
IF DInput.CV01顶升故障检测  AND   Alarm_Code=0 THEN
	Alarm_Code:=21;
END_IF;

(*入库输送线变频器电机故障*)
IF DInput.Bx02顶升故障检测  AND   Alarm_Code=0 THEN
	Alarm_Code:=22;
END_IF;

(*出库口顶升变频器电机故障*)
IF DInput.Bx04输送故障检测 AND   Alarm_Code=0 THEN
	Alarm_Code:=23;
END_IF;

(*出库货叉顶升变频器电机故障*)
IF DInput.Bx03顶升故障检测  AND   Alarm_Code=0 THEN
	Alarm_Code:=24;
END_IF;

(*出库输送线变频器电机故障*)
IF DInput.Bx04顶升故障检测  AND   Alarm_Code=0 THEN
	Alarm_Code:=25;
END_IF;

(*RFID通讯故障*)	
(*IF M340 AND Alarm_Code=0 THEN
	Alarm_Code:=26;
END_IF;
IF M341 AND Alarm_Code=0 THEN
	Alarm_Code:=27;
END_IF;*)

(*A01通讯故障*)	
(*IF M707 AND Alarm_Code=0 THEN
	Alarm_Code:=28;
END_IF;*)

(*初始化失败*)	
 OUT_T(Device_Initialization,TC12,150);
IF TS12 AND Alarm_Code=0 THEN
	Alarm_Code:=29;
END_IF;

(*弹出报警画面*)
IF Alarm_Code<>0 AND NOT Alarm_Rising THEN
     HMI_Screen:=5;
END_IF;
Alarm_Rising:=Alarm_Code<>0 ;

(*故障复位*)
IF (DInput.Alarm_Reset OR HMI.Alarm_Reset OR CCLink_W_Control_Bit.Alarm_Reset) AND Alarm_Code<>0 THEN
	Axle_IN_Sew_Control_Bit.Alarm_Reset:=TRUE;
	Axle_OUT_Sew_Control_Bit.Alarm_Reset:=TRUE;
	Alarm_Code:=0;
	Deliver_In.Step1:=0;
	Deliver_OUT.Step1:=0;
	Deliver_In.Current_Task_Status:=0;
	Deliver_OUT.Current_Task_Status:=0;
	DOutput.CV2_Jacking_Fork_Reset:=TRUE;
	DOutput.CV2_Jacking_Reset:=TRUE;
	DOutput.CV1_Jacking_Fork_Reset:=TRUE;
	DOutput.CV1_Jacking_Reset:=TRUE;
	DOutput.CV1_Conveying_Reset:=TRUE;
	DOutput.CV2_Conveying_Reset:=TRUE;
ELSE
	Axle_IN_Sew_Control_Bit.Alarm_Reset:=FALSE;
	Axle_OUT_Sew_Control_Bit.Alarm_Reset:=FALSE;
	DOutput.CV2_Jacking_Fork_Reset:=FALSE;
	DOutput.CV2_Jacking_Reset:=FALSE;
	DOutput.CV1_Jacking_Fork_Reset:=FALSE;
	DOutput.CV1_Jacking_Reset:=FALSE;
	DOutput.CV1_Conveying_Reset:=FALSE;
	DOutput.CV2_Conveying_Reset:=FALSE;
END_IF;

(*警告码*)
(*CV1: 1： 无法匹配csv计划文件，2：入库托盘重复，3：自动化仓库库满等待入库，4：出库任务取消
   CV2: 1：计划不满足，2：RFID不匹配，3：计划不满足，且RFID不匹配，4：出库任务取消 *)
IF CCLink_W.CV1_RFID_Alarm=1  AND Mode=0 THEN
		Warning_Code:=1;
		M720:=TRUE;
END_IF;
IF CCLink_W.CV1_RFID_Alarm=2 AND Mode=0 THEN
		Warning_Code:=2;
		M721:=TRUE;
END_IF;
IF CCLink_W.CV1_RFID_Alarm=3 AND Mode=0 THEN
		Warning_Code:=3;
		M722:=TRUE;
END_IF;
IF CCLink_W.CV1_RFID_Alarm=4  AND Mode=0 THEN
		Warning_Code:=4;
		M723:=TRUE;
END_IF;

IF CCLink_W.CV2_RFID_Alarm=1  AND Mode=0 THEN
		Warning_Code:=11;
		M730:=TRUE;
END_IF;
IF CCLink_W.CV2_RFID_Alarm=2  AND Mode=0 THEN
		Warning_Code:=12;
		M731:=TRUE;
END_IF;
IF CCLink_W.CV2_RFID_Alarm=3  AND Mode=0 THEN
		Warning_Code:=13;
		M732:=TRUE;
END_IF;	
IF CCLink_W.CV2_RFID_Alarm=4  AND Mode=0 THEN
		Warning_Code:=14;
		M733:=TRUE;
END_IF;	

(*IF CCLink_W.CV1_RFID_Alarm=0 THEN*)
(*IF DInput.Alarm_Reset AND Warning_Code<>0 THEN*)
IF DInput.Alarm_Reset THEN
	CCLink_W.CV1_RFID_Alarm:=0;
	Warning_Code:=0;
	K1M720:=0;
END_IF;	
(*IF CCLink_W.CV2_RFID_Alarm=0 THEN*)
(*IF DInput.Alarm_Reset AND Warning_Code<>0 THEN*)
IF DInput.Alarm_Reset THEN
	CCLink_W.CV2_RFID_Alarm:=0;
	Warning_Code:=0;
	K1M730:=0;
END_IF;
END_PROGRAM

FUNCTION_BLOCK Store
(*入库台初始化*)
IF (Mode>1   OR Alarm_Code<>0 ) AND Device_Initialization=FALSE THEN
	Deliver_In. 入库口顶升下降控制:=FALSE;
	Deliver_In. 入库口顶升上升控制:=FALSE;
	Deliver_In. 货叉顶升上升控制:=FALSE;
	Deliver_In. 货叉顶升下降控制:=FALSE;
	Deliver_In. 输送线控制:=FALSE;
    Deliver_In. 输送线低速控制:=FALSE;
    Deliver_In.货叉伸出控制:=FALSE;
    Deliver_In.货叉缩回控制:=FALSE;
END_IF;

(*初始化*)
IF DOutput.Start_Button_Indicator_Light AND NOT Start_Rising THEN
	Device_Initialization:=TRUE;
END_IF;
Start_Rising:=DOutput.Start_Button_Indicator_Light;
IF Device_Initialization AND  DOutput.Start_Button_Indicator_Light THEN
	IF Deliver_In. 入库口顶升下限检测=FALSE AND Deliver_In. 入库口物料检测=FALSE THEN
		Deliver_In. 入库口顶升下降控制:=TRUE;
	END_IF;
	IF Deliver_In. 货叉顶升下限检测=FALSE THEN
		Deliver_In. 货叉顶升下降控制:=TRUE;
	END_IF;
	IF Deliver_Out.出库口顶升上限检测=FALSE AND Deliver_Out.出库口物料检测=FALSE THEN
		Deliver_Out.出库口顶升上升控制:=TRUE;
	END_IF;
	IF Deliver_Out.货叉顶升下限检测=FALSE THEN
		Deliver_Out.货叉顶升下降控制:=TRUE;
	END_IF;
	IF Cv1_Fork_Zero_Pos=FALSE THEN
		Deliver_In.货叉缩回控制:=TRUE;
	END_IF;
	IF Cv2_Fork_Zero_Pos=FALSE THEN
		Deliver_Out.货叉缩回控制:=TRUE;
	END_IF;
	IF  Deliver_In. 入库口顶升下限检测 AND Deliver_In. 货叉顶升下限检测 AND 
		 Deliver_Out.出库口顶升上限检测 AND Deliver_Out.货叉顶升下限检测 AND 
		 Cv1_Fork_Zero_Pos AND Cv2_Fork_Zero_Pos THEN
		 Deliver_In. 入库口顶升下降控制:=FALSE;
		 Deliver_In. 货叉顶升下降控制:=FALSE;
		 Deliver_Out.出库口顶升上升控制:=FALSE;
		 Deliver_Out.货叉顶升下降控制:=FALSE;
		 Deliver_In.货叉缩回控制:=FALSE;
		 Deliver_Out.货叉缩回控制:=FALSE;
		 Initialization_Done:=TRUE;
		 Device_Initialization:=FALSE;
	END_IF;
END_IF;
IF DOutput.Start_Button_Indicator_Light=FALSE THEN
	Initialization_Done:=FALSE;
	Device_Initialization:=FALSE;
END_IF;

(*报警*)
IF Alarm_Code<>0 AND Deliver_In.Step1<>0 THEN
	Deliver_In.Step1:=0;
	Deliver_In.Current_Task_Status:=3;
END_IF;

(*堆垛机取货完成*)
IF Deliver_In. 入库口顶升下限检测=FALSE AND Deliver_In. 入库口物料检测=FALSE AND NOT CCLink_W_Control_Bit.Stacker_Picking_Goods_Mark AND Stacker_Picking_Goods AND Mode<=1 THEN
		Deliver_In. 入库口顶升下降控制:=TRUE;
END_IF;
Stacker_Picking_Goods:=CCLink_W_Control_Bit.Stacker_Picking_Goods_Mark;
IF Deliver_In. 入库口顶升下限检测 THEN
	Deliver_In. 入库口顶升下降控制:=FALSE;
END_IF;

(*货叉到入库口*)
(*联机*)
 IF Master_R.Device_Status=1  AND Mode=0  AND CCLink_W.CV1_TaskID <>Deliver_In.Current_TaskID AND CCLink_W.CV1_TaskID<>0 
 	AND Deliver_In.Step1=0  AND Alarm_Code=0  AND Deliver_In. 货叉位置物料检测 AND Deliver_In. 入库口物料检测=FALSE  AND Master_R.CV1_Current_RFID<>'' THEN
 	
	  Deliver_In.Current_TaskID:=CCLink_W.CV1_TaskID ;
	  Deliver_In.Current_Task_Status:=1;
	  Deliver_In.Step1:=1;
	  CCLink_R.CV1_AGVPick_Goods_Done:=0;
END_IF; 
(*单机*)
 IF Master_R.Device_Status=1  AND Mode=1  AND SingleID_Cv1 <>Deliver_In.Current_TaskID  AND SingleID_Cv1<>0
 	AND Deliver_In.Step1=0  AND Alarm_Code=0  AND Deliver_In. 货叉位置物料检测 AND Deliver_In. 入库口物料检测=FALSE THEN
 	
	  Deliver_In.Current_TaskID:=SingleID_Cv1 ;
	  Deliver_In.Current_Task_Status:=1;
	  Deliver_In.Step1:=1;
	  CCLink_R.CV1_AGVPick_Goods_Done:=0;
END_IF; 

(*流程开始*)
IF Deliver_In.Step1=1 AND Deliver_In. 货叉位置物料检测 AND Deliver_In. 入库口物料检测=FALSE THEN
	IF Deliver_In. 入库口顶升下限检测=FALSE THEN
		Deliver_In. 入库口顶升下降控制:=TRUE;
	END_IF;
	IF Deliver_In. 入库口顶升下限检测  THEN
		Deliver_In. 入库口顶升下降控制:=FALSE;
		Deliver_In.Step1:=2;
	END_IF;
END_IF;

IF Deliver_In.Step1=2 AND Deliver_In. 入库口顶升下限检测 THEN
	 Deliver_In. 输送线控制:=TRUE;
	IF Deliver_In. 入库口减速检测 THEN
		Deliver_In. 输送线低速控制:=TRUE;
	END_IF;
	IF Deliver_In. 入库口物料检测 THEN
		Deliver_In. 输送线控制:=FALSE;
        Deliver_In. 输送线低速控制:=FALSE;
        Deliver_In.Step1:=3;
	END_IF;
END_IF;

IF Deliver_In.Step1=3 AND Deliver_In. 入库口物料检测  THEN
	Deliver_In. 入库口顶升上升控制:=TRUE;
     Deliver_In.Step1:=4;
END_IF;
 
IF Deliver_In.Step1=4 AND Deliver_In. 入库口顶升上限检测 THEN
	Deliver_In. 入库口顶升上升控制:=FALSE;
	Deliver_In.Current_Task_Status:=2;
    Deliver_In.Step1:=0;
    SingleID_Cv1:=0;
    CCLink_W.CV1_TaskID:=0;
END_IF;

(*AGV进入中_屏蔽光栅*)
IF DInput.Photonic1_output2 AND DInput.Photonic1_Go AND DInput.Photonic2_Go=FALSE AND DInput.Photonic3_Go=FALSE AND Deliver_In.AGV进入中=FALSE AND  Master_R.Device_Status=1 AND AGV_CVArea=FALSE THEN
	   Deliver_In.AGV进入中:=TRUE;
	   DOutput.Photonic1_Input3:=TRUE;
	   AGV_CVArea :=TRUE;
ELSIF
	  DOutput.Photonic1_Input3 AND DInput.Photonic1_Go=FALSE THEN
	  DOutput.Photonic1_Input3:=FALSE;	
END_IF;

  (*AGV到达入库口*)
  IF DInput.Photonic2_output2 AND DInput.Photonic2_Go THEN
	   Deliver_In.AGV进入中:=FALSE; 	
  END_IF;
  
Deliver_In.AGV_Go:= DInput.Photonic2_Go ;
Deliver_In.AGV_Stop_Status:= DInput.Photonic2_output2 ;
Deliver_In.AGV物料探测:=DInput.CV01AGV物料检测;
Deliver_In.AGV本体检测:=1;
DOutput.Photonic2_Input3:=Deliver_In.AGV放行;

(*AGV到货叉*)
IF Master_R.Device_Status=1  AND  Mode<=1  AND Deliver_In.AGV_Go AND Deliver_In.AGV_Stop_Status   AND Deliver_In.Step1=0  AND Alarm_Code=0 AND
	 Deliver_In.AGV物料探测 AND Deliver_In. 货叉位置物料检测=FALSE AND Deliver_In.AGV本体检测 THEN
	 
    Deliver_In.Current_Task_Status:=1;
	Deliver_In.Step1:=10;
END_IF;

IF  Deliver_In.Step1=10 AND  Deliver_In.AGV物料探测 AND Deliver_In. 货叉位置物料检测=FALSE THEN
	IF Deliver_In. 货叉顶升下限检测=FALSE THEN
		Deliver_In. 货叉顶升下降控制:=TRUE;
	END_IF;
	IF Deliver_In. 货叉顶升下限检测  THEN
		Deliver_In. 货叉顶升下降控制:=FALSE;
		Deliver_In.Step1:=11;
	END_IF;
END_IF;

IF  Deliver_In.Step1=11 AND Deliver_In. 货叉顶升下限检测 THEN
	Deliver_In.货叉伸出控制:=TRUE;
	Deliver_In.Step1:=12;
END_IF;
  
  IF  Deliver_In.Step1=12 AND Deliver_In. 货叉伸出到位 THEN
  	Deliver_In.货叉伸出控制:=FALSE;
  	Deliver_In. 货叉顶升上升控制:=TRUE;
	Deliver_In.Step1:=13;
  END_IF;
  
  IF  Deliver_In.Step1=13 AND Deliver_In. 货叉顶升上限检测 THEN
    	Deliver_In. 货叉顶升上升控制:=FALSE;
    	Deliver_In.货叉缩回控制:=TRUE;
    	Deliver_In.Step1:=14;
  END_IF;
  
  IF Deliver_In.Step1=14 AND Deliver_In. 货叉缩回到位 THEN
  	Deliver_In.货叉缩回控制:=FALSE;
  	Deliver_In. 货叉顶升下降控制:=TRUE;
    Deliver_In.Step1:=15;
  END_IF;
    	
IF Deliver_In.Step1=15  AND Deliver_In. 货叉顶升下限检测 THEN
	    Deliver_In. 入库口顶升下降控制:=FALSE;
		Deliver_In. 货叉顶升下降控制:=FALSE;
		Deliver_In.Current_Task_Status:=2;
		Deliver_In.Step1:=0;
		CCLink_R.CV1_AGVPick_Goods_Done:=1001;
		(*AGV放行*)
        Deliver_In.AGV放行:=TRUE;
END_IF;

(*AGV入库台 放行完成*)
IF Deliver_In.AGV放行 AND DInput.Photonic2_Go=FALSE THEN
	Deliver_In.AGV放行:=FALSE;
END_IF;
END_FUNCTION_BLOCK

FUNCTION_BLOCK Outbound
(*出库台初始化*)
IF (Mode>1 OR  Deliver_Out.Step1=0  OR Alarm_Code<>0 )AND Device_Initialization=FALSE THEN
	Deliver_Out.出库口顶升下降控制:=FALSE;
	Deliver_Out.出库口顶升上升控制:=FALSE;
	Deliver_Out.货叉顶升上升控制:=FALSE;
	Deliver_Out.货叉顶升下降控制:=FALSE;
	Deliver_Out.输送线控制:=FALSE;
    Deliver_Out.输送线低速控制:=FALSE;
    Deliver_Out.货叉伸出控制:=FALSE;
    Deliver_Out.货叉缩回控制:=FALSE;
	CCLink_R.CV2_AGVPurpose:=0;
END_IF;

(*报警*)
IF Alarm_Code<>0 AND Deliver_Out.Step1<>0 THEN
	Deliver_Out.Step1:=0;
	Deliver_OUT.Current_Task_Status:=3;
END_IF;

(*出库口到货叉*)
(*联机*)
IF Master_R.Device_Status=1  AND Mode=0 AND  CCLink_W.CV2_TaskID<>Deliver_Out.Current_TaskID AND CCLink_W.CV2_TaskID<>0 
	AND Deliver_Out.Step1=0  AND Alarm_Code=0  AND Deliver_Out.货叉位置物料检测=FALSE AND Deliver_Out.出库口物料检测 THEN
	Deliver_Out.Current_TaskID:=CCLink_W.CV2_TaskID;
	Deliver_OUT.Current_Task_Status:=1;
	Deliver_Out.Step1:=1;
END_IF;
(*单机*)
IF Master_R.Device_Status=1  AND Mode=1 AND  SingleID_Cv2<>Deliver_Out.Current_TaskID AND SingleID_Cv2<>0
	 AND Deliver_Out.Step1=0  AND Alarm_Code=0  AND Deliver_Out.货叉位置物料检测=FALSE AND Deliver_Out.出库口物料检测 THEN
	Deliver_Out.Current_TaskID:=SingleID_Cv2;
	Deliver_OUT.Current_Task_Status:=1;
	Deliver_Out.Step1:=1;
END_IF;

(*流程开始*)
IF Deliver_Out.Step1=1 AND Deliver_Out.货叉位置物料检测=FALSE AND Deliver_Out.出库口物料检测 THEN
		Deliver_Out.出库口顶升下降控制:=TRUE;
		Deliver_Out.Step1:=2;
END_IF;

IF Deliver_Out.Step1=2 AND Deliver_Out.出库口顶升下限检测 THEN
	Deliver_Out.出库口顶升下降控制:=FALSE;
	IF Deliver_Out.货叉顶升下限检测=FALSE THEN
	Deliver_Out.货叉顶升下降控制:=TRUE;
	END_IF;
	IF Deliver_Out.货叉顶升下限检测 THEN
		Deliver_Out.货叉顶升下降控制:=FALSE;
	    Deliver_Out.输送线控制:=TRUE;
	    Deliver_Out.Step1:=3;
	END_IF;
END_IF;

IF Deliver_Out.Step1=3   THEN
	IF Deliver_Out.货叉位置减速检测 THEN
		Deliver_Out.输送线低速控制:=TRUE;
	END_IF;
	IF Deliver_Out.货叉位置物料检测 THEN
		Deliver_Out.输送线控制:=FALSE;
        Deliver_Out.输送线低速控制:=FALSE;
       Deliver_Out. Step1:=4;
	END_IF;
END_IF;

IF Deliver_Out.Step1=4 AND Deliver_Out.出库口物料检测=FALSE THEN
	Deliver_Out.出库口顶升上升控制:=TRUE;
	Deliver_Out.Step1:=5;
END_IF;
 
IF Deliver_Out.Step1=5 AND Deliver_Out.出库口顶升上限检测 THEN
	Deliver_Out.出库口顶升上升控制:=FALSE;
	Deliver_OUT.Current_Task_Status:=2;
   Deliver_Out. Step1:=0;
   SingleID_Cv2:=0;
   CCLink_W.CV2_TaskID:=0;
END_IF;

 Deliver_Out.AGV_Go:=DInput.Photonic3_Go ;
Deliver_Out.AGV_Stop_Status:=DInput.Photonic3_output2 ;
Deliver_Out.AGV本体检测:=1 ;
Deliver_Out.AGV物料探测:=DInput.Bx03AGV物料检测;
DOutput.Photonic3_Input3:=Deliver_Out.AGV放行;
(*货叉到AGV*)
(*联机*)
IF Master_R.Device_Status=1  AND Mode=0 AND ((CCLink_W.CV2_Allow_GoodsToAGV<>0  AND CCLink_R.CV2_AGVPurpose<>CCLink_W.CV2_Allow_GoodsToAGV )OR W42=1 )AND Deliver_Out.AGV_Go AND Deliver_Out.AGV_Stop_Status   AND 
	Deliver_Out.Step1=0  AND Alarm_Code=0 AND Deliver_Out.AGV物料探测=FALSE  AND Deliver_Out.货叉位置物料检测 AND Deliver_Out.AGV本体检测 AND Master_R.CV2_Current_RFID<>''  THEN
    Deliver_OUT.Current_Task_Status:=1;
	Deliver_Out.Step1:=10;
	CCLink_R.CV2_AGVPurpose:=CCLink_W.CV2_Allow_GoodsToAGV;
END_IF;
(*单机*)
IF Master_R.Device_Status=1  AND Mode=1 AND (SingleAGVPurpose_Cv2<>0  OR W42=1 ) AND Deliver_Out.AGV_Go AND Deliver_Out.AGV_Stop_Status   AND 
	Deliver_Out.Step1=0  AND Alarm_Code=0 AND Deliver_Out.AGV物料探测=FALSE  AND Deliver_Out.货叉位置物料检测 AND Deliver_Out.AGV本体检测 THEN
    Deliver_OUT.Current_Task_Status:=1;
	Deliver_Out.Step1:=10;
	CCLink_R.CV2_AGVPurpose:=SingleAGVPurpose_Cv2;
	SingleAGVPurpose_Cv2:=0;
END_IF;

IF  Deliver_Out.Step1=10 AND  Deliver_Out.AGV物料探测=FALSE AND Deliver_Out.货叉位置物料检测 THEN
	IF Cv2_Fork_Zero_Pos=FALSE THEN
		Deliver_Out.货叉缩回控制:=TRUE;
		Deliver_Out.Step1:=11;
	END_IF ;
	IF Cv2_Fork_Zero_Pos THEN
		Deliver_Out.货叉缩回控制:=FALSE;
		Deliver_Out.Step1:=11;
	END_IF ;
END_IF;

IF  	Deliver_Out.Step1=11 AND Deliver_Out.货叉缩回到位 THEN
	    Deliver_Out.货叉缩回控制:=FALSE;
		Deliver_Out.货叉顶升上升控制:=TRUE;
		CCLink_R.CV2_AGVReleaseGoods_Done:=0;
		Deliver_Out.Step1:=12;
END_IF;

IF  Deliver_Out.Step1=12 AND Deliver_Out.货叉顶升上限检测 THEN
	Deliver_Out.货叉顶升上升控制:=FALSE;
	Deliver_Out.货叉伸出控制:=TRUE;
	Deliver_Out.Step1:=13;
END_IF;
  
  IF  Deliver_Out.Step1=13 AND Deliver_Out.货叉伸出到位 THEN
  	Deliver_Out.货叉伸出控制:=FALSE;
  	Deliver_Out.货叉顶升下降控制:=TRUE;
	Deliver_Out.Step1:=14;
  END_IF;
  
  IF  Deliver_Out.Step1=14 AND Deliver_Out.货叉顶升下限检测 THEN
    	Deliver_Out.货叉顶升下降控制:=FALSE;
    	Deliver_Out.货叉缩回控制:=TRUE;
    	Deliver_Out.Step1:=15;
  END_IF;
  
  IF Deliver_Out.Step1=15 AND Deliver_Out.货叉缩回到位 THEN
  	Deliver_Out.货叉缩回控制:=FALSE;
  	Deliver_OUT.Current_Task_Status:=2;
	Deliver_Out.Step1:=0;
	CCLink_R.CV2_AGVReleaseGoods_Done:=1;	
	SingleAGVPurpose_Cv2:=0;
  END_IF;
  
  (*AGV放行*)
IF  CCLink_R.CV2_AGVReleaseGoods_Done=1 AND  Deliver_Out.AGV_Go AND Deliver_Out.AGV物料探测 AND Deliver_Out.AGV本体检测 THEN
	  Deliver_Out.AGV放行:=TRUE;
	   Deliver_Out.AGVl离开中:=TRUE;
ELSIF
	  CCLink_R.CV2_AGVReleaseGoods_Done=1 AND  Deliver_Out.AGV_Go=FALSE  THEN
	   Deliver_Out.AGV放行:=FALSE;
	  CCLink_R.CV2_AGVReleaseGoods_Done:=0;
	  CCLink_R.CV2_AGVPurpose:=0;
END_IF;

(*AGV已离开_打开光栅*)
IF DInput.Photonic4_output2 AND DInput.Photonic4_Go THEN
	   Deliver_Out.AGVl离开中:=FALSE;
	   DOutput.Photonic4_Input3:=TRUE;
	   AGV_CVArea :=FALSE;
ELSIF
	  DOutput.Photonic4_Input3 AND DInput.Photonic4_Go=FALSE THEN
	  DOutput.Photonic4_Input3:=FALSE;	
END_IF;

IF  AGV_CVArea AND DInput.Photonic3_Go =FALSE AND DInput.Photonic2_Go =FALSE AND Mode>1 THEN
	AGV_CVArea :=FALSE;
END_IF;
END_FUNCTION_BLOCK

PROGRAM Manual
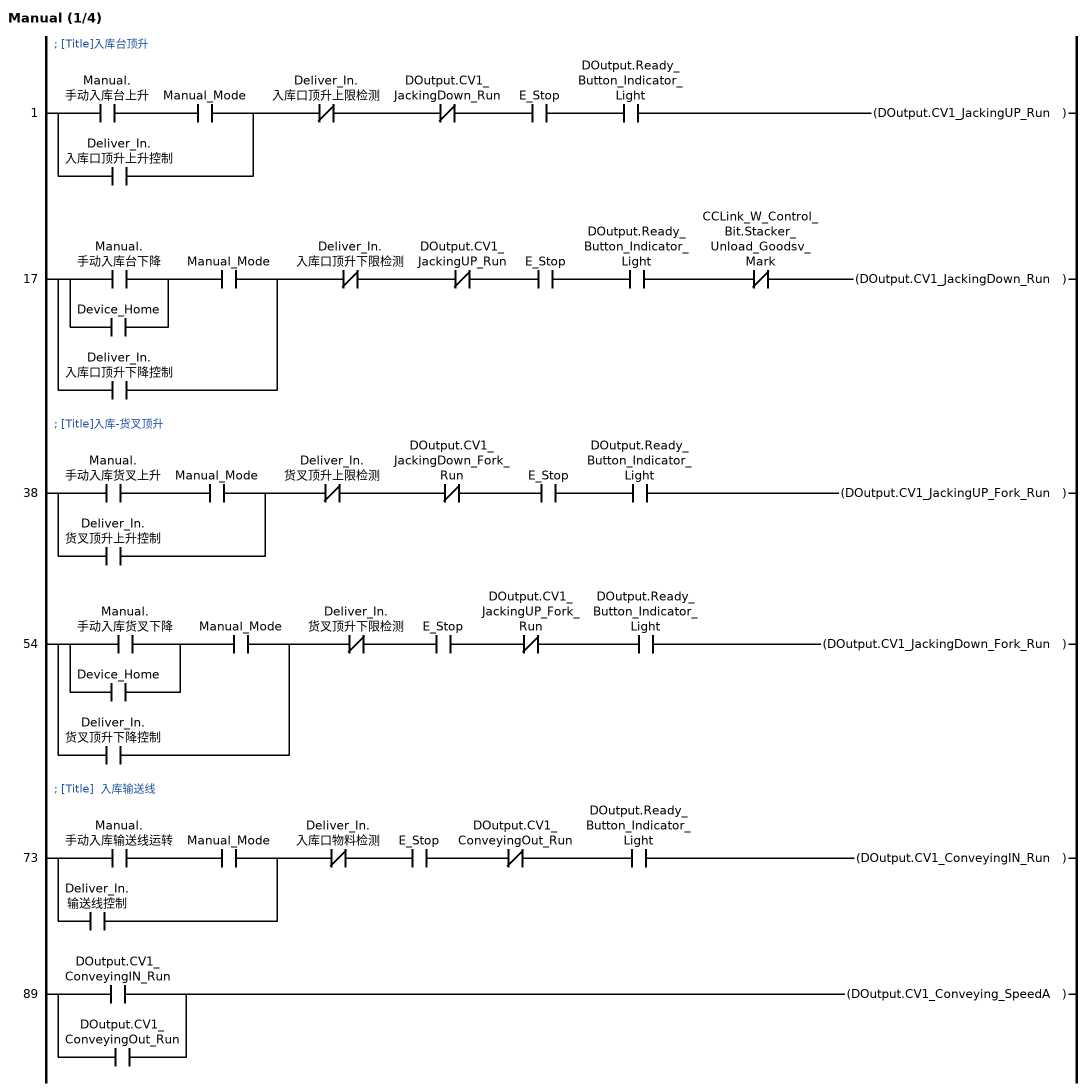
; [Title]入库台顶升
1     LD      Manual.手动入库台上升
      AND     Manual_Mode
      OR      Deliver_In.入库口顶升上升控制
      ANI     Deliver_In.入库口顶升上限检测
      ANI     DOutput.CV1_JackingDown_Run
      AND     E_Stop
      AND     DOutput.Ready_Button_Indicator_Light
      OUT     DOutput.CV1_JackingUP_Run
17    LD      Manual.手动入库台下降
      OR      Device_Home
      AND     Manual_Mode
      OR      Deliver_In.入库口顶升下降控制
      ANI     Deliver_In.入库口顶升下限检测
      ANI     DOutput.CV1_JackingUP_Run
      AND     E_Stop
      AND     DOutput.Ready_Button_Indicator_Light
      ANI     CCLink_W_Control_Bit.Stacker_Unload_Goodsv_Mark
      OUT     DOutput.CV1_JackingDown_Run
; [Title]入库-货叉顶升
38    LD      Manual.手动入库货叉上升
      AND     Manual_Mode
      OR      Deliver_In.货叉顶升上升控制
      ANI     Deliver_In.货叉顶升上限检测
      ANI     DOutput.CV1_JackingDown_Fork_Run
      AND     E_Stop
      AND     DOutput.Ready_Button_Indicator_Light
      OUT     DOutput.CV1_JackingUP_Fork_Run
54    LD      Manual.手动入库货叉下降
      OR      Device_Home
      AND     Manual_Mode
      OR      Deliver_In.货叉顶升下降控制
      ANI     Deliver_In.货叉顶升下限检测
      AND     E_Stop
      ANI     DOutput.CV1_JackingUP_Fork_Run
      AND     DOutput.Ready_Button_Indicator_Light
      OUT     DOutput.CV1_JackingDown_Fork_Run
; [Title]  入库输送线
73    LD      Manual.手动入库输送线运转
      AND     Manual_Mode
      OR      Deliver_In.输送线控制
      ANI     Deliver_In.入库口物料检测
      AND     E_Stop
      ANI     DOutput.CV1_ConveyingOut_Run
      AND     DOutput.Ready_Button_Indicator_Light
      OUT     DOutput.CV1_ConveyingIN_Run
89    LD      DOutput.CV1_ConveyingIN_Run
      OR      DOutput.CV1_ConveyingOut_Run
      OUT     DOutput.CV1_Conveying_SpeedA
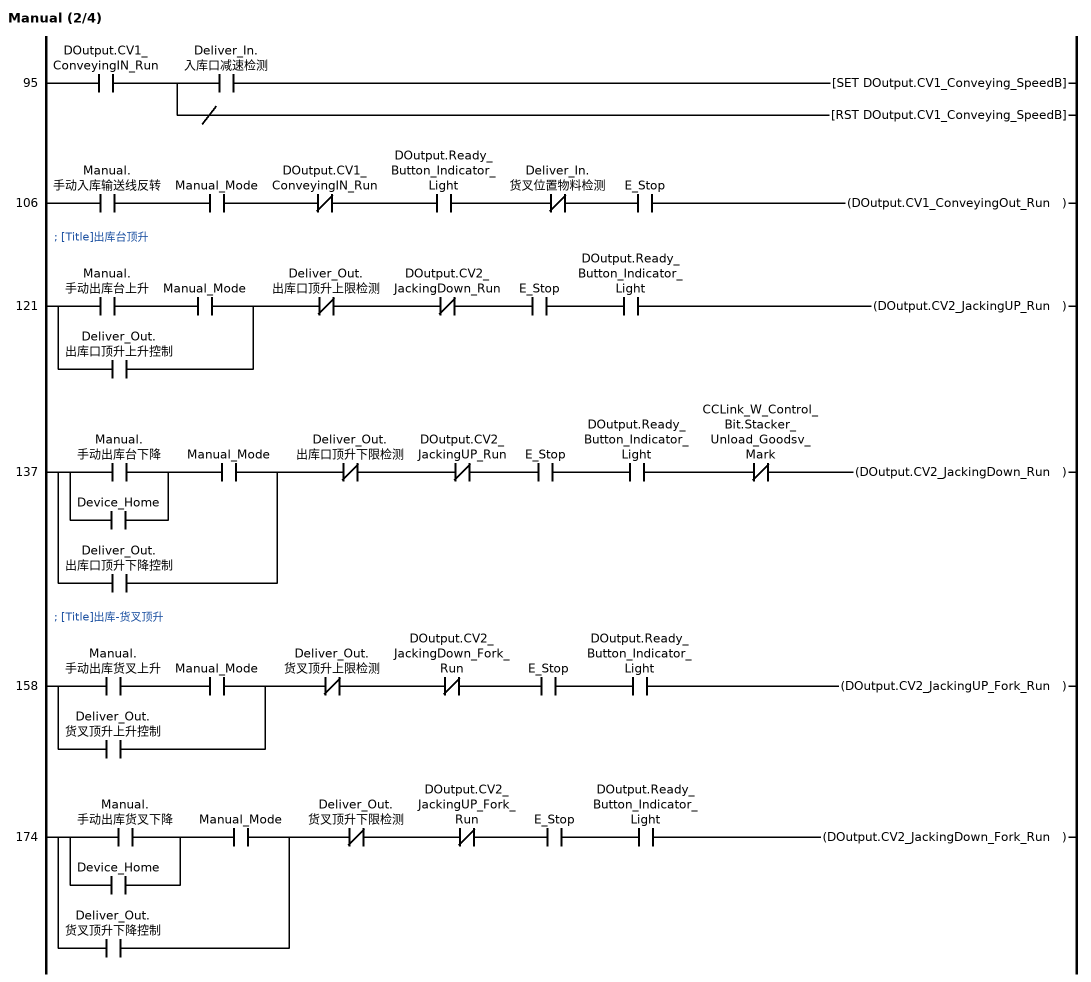
95    LD      DOutput.CV1_ConveyingIN_Run
      MPS
      AND     Deliver_In.入库口减速检测
      SET     DOutput.CV1_Conveying_SpeedB
      MPP
      INV
      RST     DOutput.CV1_Conveying_SpeedB
106   LD      Manual.手动入库输送线反转
      AND     Manual_Mode
      ANI     DOutput.CV1_ConveyingIN_Run
      AND     DOutput.Ready_Button_Indicator_Light
      ANI     Deliver_In.货叉位置物料检测
      AND     E_Stop
      OUT     DOutput.CV1_ConveyingOut_Run
; [Title]出库台顶升
121   LD      Manual.手动出库台上升
      AND     Manual_Mode
      OR      Deliver_Out.出库口顶升上升控制
      ANI     Deliver_Out.出库口顶升上限检测
      ANI     DOutput.CV2_JackingDown_Run
      AND     E_Stop
      AND     DOutput.Ready_Button_Indicator_Light
      OUT     DOutput.CV2_JackingUP_Run
137   LD      Manual.手动出库台下降
      OR      Device_Home
      AND     Manual_Mode
      OR      Deliver_Out.出库口顶升下降控制
      ANI     Deliver_Out.出库口顶升下限检测
      ANI     DOutput.CV2_JackingUP_Run
      AND     E_Stop
      AND     DOutput.Ready_Button_Indicator_Light
      ANI     CCLink_W_Control_Bit.Stacker_Unload_Goodsv_Mark
      OUT     DOutput.CV2_JackingDown_Run
; [Title]出库-货叉顶升
158   LD      Manual.手动出库货叉上升
      AND     Manual_Mode
      OR      Deliver_Out.货叉顶升上升控制
      ANI     Deliver_Out.货叉顶升上限检测
      ANI     DOutput.CV2_JackingDown_Fork_Run
      AND     E_Stop
      AND     DOutput.Ready_Button_Indicator_Light
      OUT     DOutput.CV2_JackingUP_Fork_Run
174   LD      Manual.手动出库货叉下降
      OR      Device_Home
      AND     Manual_Mode
      OR      Deliver_Out.货叉顶升下降控制
      ANI     Deliver_Out.货叉顶升下限检测
      ANI     DOutput.CV2_JackingUP_Fork_Run
      AND     E_Stop
      AND     DOutput.Ready_Button_Indicator_Light
      OUT     DOutput.CV2_JackingDown_Fork_Run
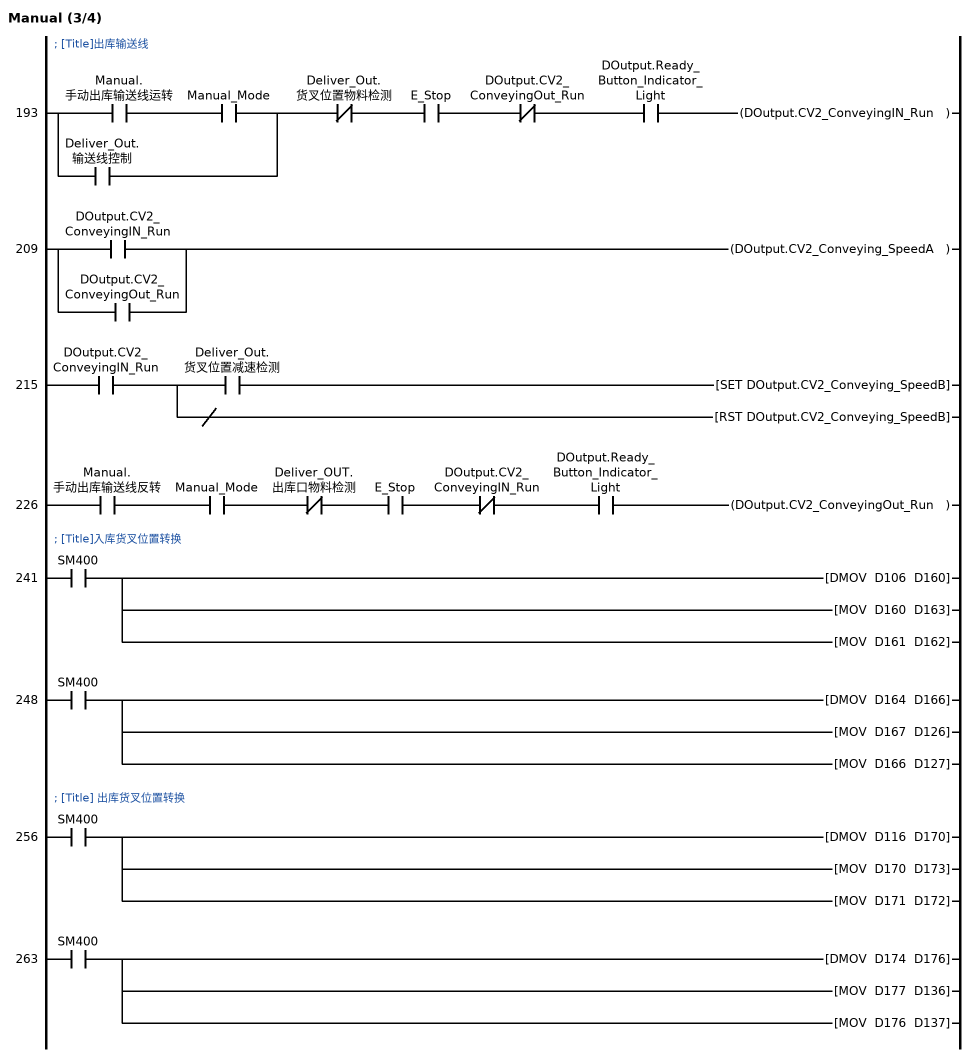
; [Title]出库输送线
193   LD      Manual.手动出库输送线运转
      AND     Manual_Mode
      OR      Deliver_Out.输送线控制
      ANI     Deliver_Out.货叉位置物料检测
      AND     E_Stop
      ANI     DOutput.CV2_ConveyingOut_Run
      AND     DOutput.Ready_Button_Indicator_Light
      OUT     DOutput.CV2_ConveyingIN_Run
209   LD      DOutput.CV2_ConveyingIN_Run
      OR      DOutput.CV2_ConveyingOut_Run
      OUT     DOutput.CV2_Conveying_SpeedA
215   LD      DOutput.CV2_ConveyingIN_Run
      MPS
      AND     Deliver_Out.货叉位置减速检测
      SET     DOutput.CV2_Conveying_SpeedB
      MPP
      INV
      RST     DOutput.CV2_Conveying_SpeedB
226   LD      Manual.手动出库输送线反转
      AND     Manual_Mode
      ANI     Deliver_OUT.出库口物料检测
      AND     E_Stop
      ANI     DOutput.CV2_ConveyingIN_Run
      AND     DOutput.Ready_Button_Indicator_Light
      OUT     DOutput.CV2_ConveyingOut_Run
; [Title]入库货叉位置转换
241   LD      SM400
      DMOV    D106 D160
      MOV     D160 D163
      MOV     D161 D162
248   LD      SM400
      DMOV    D164 D166
      MOV     D167 D126
      MOV     D166 D127
; [Title] 出库货叉位置转换
256   LD      SM400
      DMOV    D116 D170
      MOV     D170 D173
      MOV     D171 D172
263   LD      SM400
      DMOV    D174 D176
      MOV     D177 D136
      MOV     D176 D137
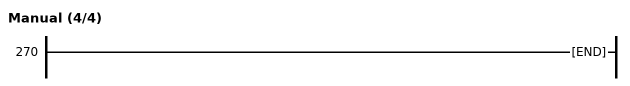
270   END
END_PROGRAM

PROGRAM drive
VAR
  RFID1 : INT;
  RFID2 : INT;
  __IST_44a547fe69a44295 : I+ST_44a547fe69a44295;
  RFID3 : INT;
  RFID4 : INT;
  RFID5 : INT;
  RFID6 : INT;
  __IST_122ae8440b094ab7 : I+ST_122ae8440b094ab7;
  RFID11 : INT;
  RFID12 : INT;
  RFID13 : INT;
  RFID14 : INT;
  RFID15 : INT;
  RFID16 : INT;
  Parse_Done_Cv1 : BOOL;
  Parse_Done_Cv2 : BOOL;
END_VAR
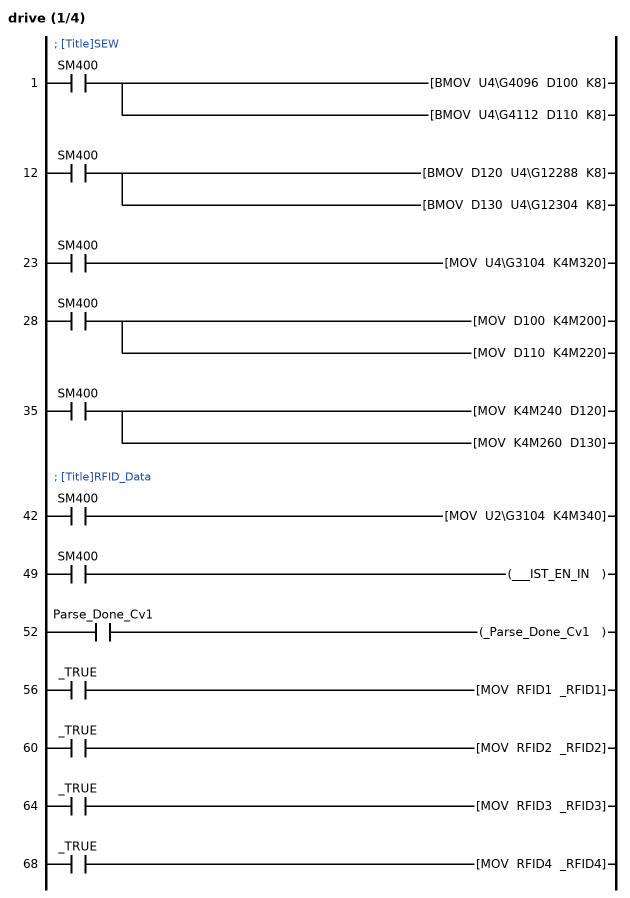
; [Title]SEW
1     LD      SM400
      BMOV    U4\G4096 D100 K8
      BMOV    U4\G4112 D110 K8
12    LD      SM400
      BMOV    D120 U4\G12288 K8
      BMOV    D130 U4\G12304 K8
23    LD      SM400
      MOV     U4\G3104 K4M320
28    LD      SM400
      MOV     D100 K4M200
      MOV     D110 K4M220
35    LD      SM400
      MOV     K4M240 D120
      MOV     K4M260 D130
; [Title]RFID_Data
42    LD      SM400
      MOV     U2\G3104 K4M340
; FB BLK START I+ST_44a547fe69a44295(__IST_44a547fe69a44295)
49    LD      SM400
      OUT     ___IST_EN_IN
52    LD      Parse_Done_Cv1
      OUT     _Parse_Done_Cv1
56    LD      _TRUE
      MOV     RFID1 _RFID1
60    LD      _TRUE
      MOV     RFID2 _RFID2
64    LD      _TRUE
      MOV     RFID3 _RFID3
68    LD      _TRUE
      MOV     RFID4 _RFID4
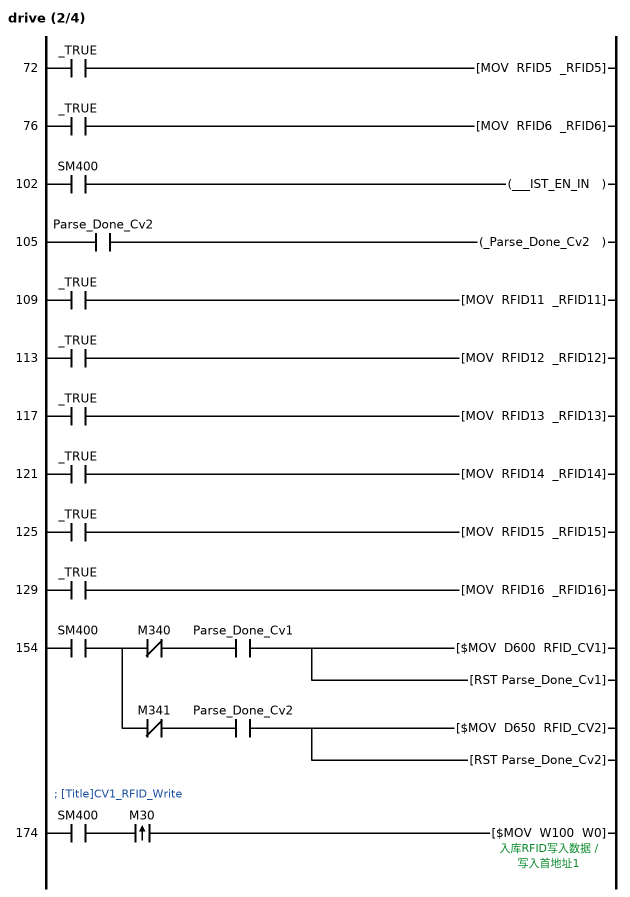
72    LD      _TRUE
      MOV     RFID5 _RFID5
76    LD      _TRUE
      MOV     RFID6 _RFID6
; FB START
; FB_NAME I+ST_44a547fe69a44295
; INSTANCE_NAME __IST_44a547fe69a44295
; FB IN_B:__IST_EN_IN
; FB OUT___IST_EN_OUT:B
; FB IN_B:Parse_Done_Cv1
; FB OUT_Parse_Done_Cv1:B
; FB IN_W:RFID1
; FB OUT_RFID1:W
; FB IN_W:RFID2
; FB OUT_RFID2:W
; FB IN_W:RFID3
; FB OUT_RFID3:W
; FB IN_W:RFID4
; FB OUT_RFID4:W
; FB IN_W:RFID5
; FB OUT_RFID5:W
; FB IN_W:RFID6
; FB OUT_RFID6:W
; FB END
; FB BLK END
; FB BLK START I+ST_122ae8440b094ab7(__IST_122ae8440b094ab7)
102   LD      SM400
      OUT     ___IST_EN_IN
105   LD      Parse_Done_Cv2
      OUT     _Parse_Done_Cv2
109   LD      _TRUE
      MOV     RFID11 _RFID11
113   LD      _TRUE
      MOV     RFID12 _RFID12
117   LD      _TRUE
      MOV     RFID13 _RFID13
121   LD      _TRUE
      MOV     RFID14 _RFID14
125   LD      _TRUE
      MOV     RFID15 _RFID15
129   LD      _TRUE
      MOV     RFID16 _RFID16
; FB START
; FB_NAME I+ST_122ae8440b094ab7
; INSTANCE_NAME __IST_122ae8440b094ab7
; FB IN_B:__IST_EN_IN
; FB OUT___IST_EN_OUT:B
; FB IN_B:Parse_Done_Cv2
; FB OUT_Parse_Done_Cv2:B
; FB IN_W:RFID11
; FB OUT_RFID11:W
; FB IN_W:RFID12
; FB OUT_RFID12:W
; FB IN_W:RFID13
; FB OUT_RFID13:W
; FB IN_W:RFID14
; FB OUT_RFID14:W
; FB IN_W:RFID15
; FB OUT_RFID15:W
; FB IN_W:RFID16
; FB OUT_RFID16:W
; FB END
; FB BLK END
154   LD      SM400
      MPS
      ANI     M340
      AND     Parse_Done_Cv1
      $MOV    D600 RFID_CV1
      RST     Parse_Done_Cv1
      MPP
      ANI     M341
      AND     Parse_Done_Cv2
      $MOV    D650 RFID_CV2
      RST     Parse_Done_Cv2
; [Title]CV1_RFID_Write
174   LD      SM400
      ANDP    M30
      $MOV    W100 W0  ; 入库RFID写入数据 / 写入首地址1
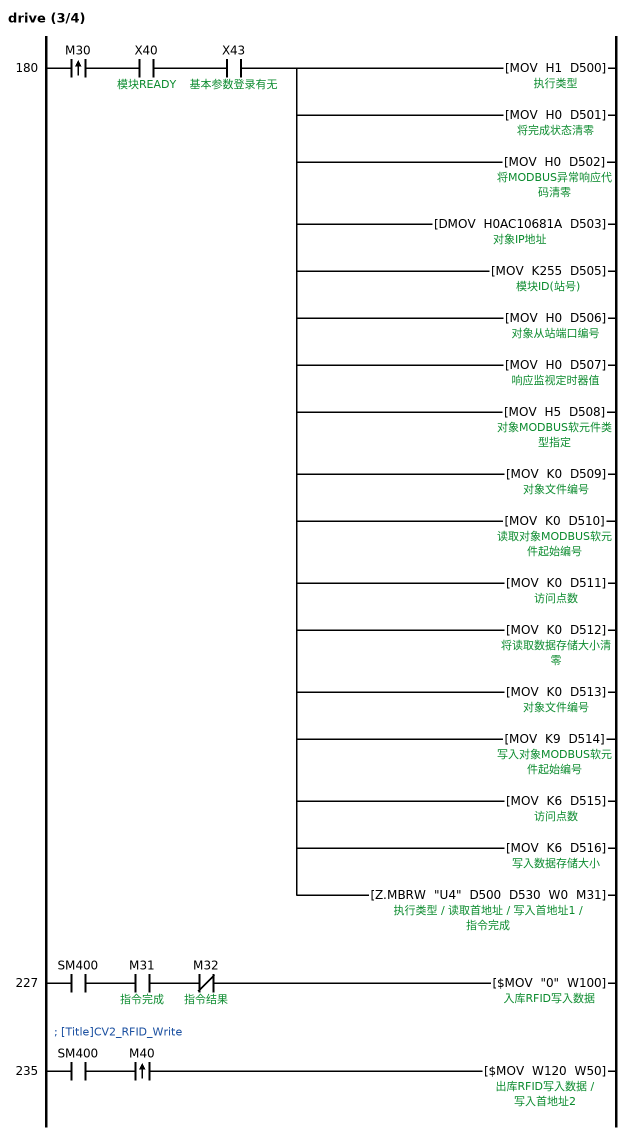
180   LDP     M30
      AND     X40  ; 模块READY
      AND     X43  ; 基本参数登录有无
      MOV     H1 D500  ; 执行类型
      MOV     H0 D501  ; 将完成状态清零
      MOV     H0 D502  ; 将MODBUS异常响应代码清零
      DMOV    H0AC10681A D503  ; 对象IP地址
      MOV     K255 D505  ; 模块ID(站号)
      MOV     H0 D506  ; 对象从站端口编号
      MOV     H0 D507  ; 响应监视定时器值
      MOV     H5 D508  ; 对象MODBUS软元件类型指定
      MOV     K0 D509  ; 对象文件编号
      MOV     K0 D510  ; 读取对象MODBUS软元件起始编号
      MOV     K0 D511  ; 访问点数
      MOV     K0 D512  ; 将读取数据存储大小清零
      MOV     K0 D513  ; 对象文件编号
      MOV     K9 D514  ; 写入对象MODBUS软元件起始编号
      MOV     K6 D515  ; 访问点数
      MOV     K6 D516  ; 写入数据存储大小
      Z.MBRW  "U4" D500 D530 W0 M31  ; 读取首地址 / 指令完成
227   LD      SM400
      AND     M31  ; 指令完成
      ANI     M32  ; 指令结果
      $MOV    "0" W100
; [Title]CV2_RFID_Write
235   LD      SM400
      ANDP    M40
      $MOV    W120 W50  ; 出库RFID写入数据 / 写入首地址2
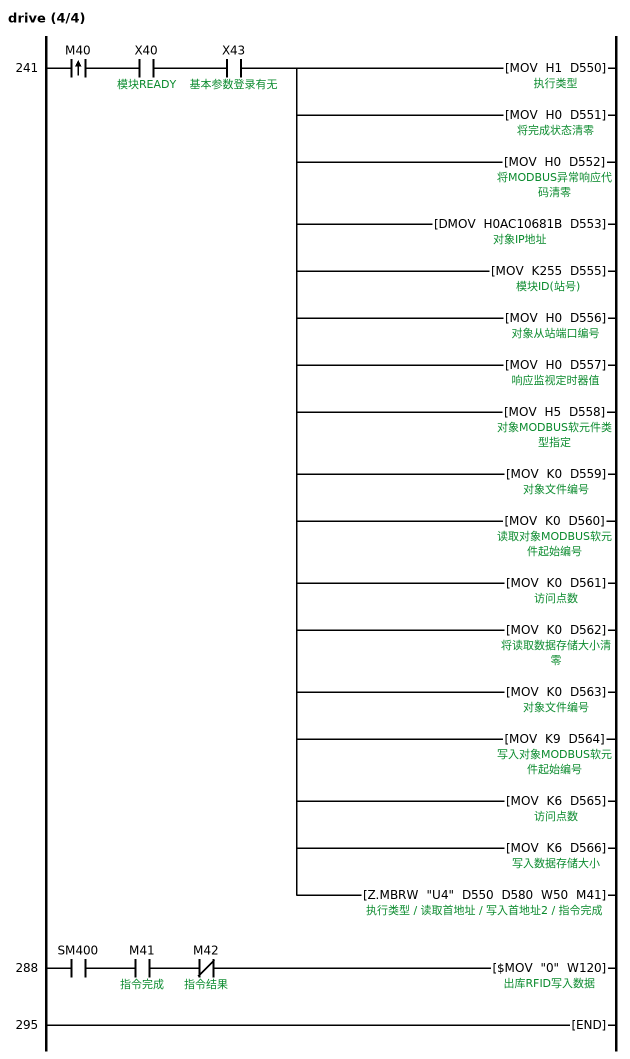
241   LDP     M40
      AND     X40  ; 模块READY
      AND     X43  ; 基本参数登录有无
      MOV     H1 D550  ; 执行类型
      MOV     H0 D551  ; 将完成状态清零
      MOV     H0 D552  ; 将MODBUS异常响应代码清零
      DMOV    H0AC10681B D553  ; 对象IP地址
      MOV     K255 D555  ; 模块ID(站号)
      MOV     H0 D556  ; 对象从站端口编号
      MOV     H0 D557  ; 响应监视定时器值
      MOV     H5 D558  ; 对象MODBUS软元件类型指定
      MOV     K0 D559  ; 对象文件编号
      MOV     K0 D560  ; 读取对象MODBUS软元件起始编号
      MOV     K0 D561  ; 访问点数
      MOV     K0 D562  ; 将读取数据存储大小清零
      MOV     K0 D563  ; 对象文件编号
      MOV     K9 D564  ; 写入对象MODBUS软元件起始编号
      MOV     K6 D565  ; 访问点数
      MOV     K6 D566  ; 写入数据存储大小
      Z.MBRW  "U4" D550 D580 W50 M41  ; 读取首地址 / 指令完成
288   LD      SM400
      AND     M41  ; 指令完成
      ANI     M42  ; 指令结果
      $MOV    "0" W120
295   END
END_PROGRAM

PROGRAM CCLink
(* 1#    RX/RY 0000-002F  RWr/RWw  0100-012F*)  (* 主站X1000(48点)  Y1000(48点)  RWw-D4000(48点)   RWr-D3000(48点)  *)
(* 2#    RX/RY 0030-005F  RWr/RWw  0130-015F*)  (* 主站X1030(48点)  Y1030(48点)  RWw-D4048(48点)   RWr-D3048(48点)  *)
(* 3#    RX/RY 0060-008F  RWr/RWw  0160-018F*)  (* 主站X1060(48点)  Y1060(48点)  RWw-D4096(48点)   RWr-D3096(48点)  *)

(* 1#    RX/RY 0000-002F  RWr/RWw  0100-012F*)  (* 主站X1000(48点)  Y1000(48点)  RWw-D3100(48点)   RWr-D3000(48点)  *)

(*Read*)
CCLink_R.Heartbeat:=TN0;
CCLink_R.Current_Mode:=Mode;
CCLink_R.Device_Status:=Master_R.Device_Status;
CCLink_R.Error_Code:=Alarm_Code;
CCLink_R.CV1_Task_Status:=Deliver_In.Current_Task_Status;
CCLink_R.CV1_Current_TaskID:=Deliver_In.Current_TaskID;

CCLink_R.CV2_Task_Status:=Deliver_OUT.Current_Task_Status;
CCLink_R.CV2_Current_TaskID:=Deliver_Out.Current_TaskID;


IF Deliver_In.入库口顶升上限检测 AND Deliver_In.入库口物料检测 AND mode=0  AND Alarm_Code=0 AND DOutput.Start_Button_Indicator_Light THEN
    CCLink_R.Stacker_PickingGoods_Status:=1;
ELSE
	CCLink_R.Stacker_PickingGoods_Status:=0;
END_IF;
IF Deliver_Out.出库口顶升上限检测 AND Deliver_Out.出库口物料检测=FALSE AND mode=0 AND Alarm_Code=0 AND DOutput.Start_Button_Indicator_Light THEN
    CCLink_R.Stacker_UnloadGoods_Status:=1;
ELSE
	CCLink_R.Stacker_UnloadGoods_Status:=0;
END_IF;

(*托盘RFID编号信息，最长12位数*)
CCLink_R.CV1_Current_RFID:=Master_R.CV1_Current_RFID;
CCLink_R.CV2_Current_RFID:=Master_R.CV2_Current_RFID;
CCLink_R.CV1_Step:=Deliver_In.Step1;
CCLink_R.CV2_Step:=Deliver_Out.Step1;

CCLink_R.CV1_Fork_Current_Pos:=DINT_TO_INT( CV1_Fork_Current_Position);
CCLink_R.CV2_Fork_Current_Pos:=DINT_TO_INT( CV2_Fork_Current_Position);

(*Rx*)
CCLink_R_Status_Bit.入库台减速检测:=Deliver_In.入库口减速检测;
CCLink_R_Status_Bit.入库台物料检测 :=Deliver_In.入库口物料检测;
CCLink_R_Status_Bit.入库货叉台物料检测:=Deliver_In.货叉位置物料检测;
CCLink_R_Status_Bit.出库台物料检测:=Deliver_OUT.出库口物料检测;
CCLink_R_Status_Bit.出库货叉台减速检测:=Deliver_OUT.货叉位置减速检测;
CCLink_R_Status_Bit.出库货叉台物料检测:=Deliver_OUT.货叉位置物料检测;
CCLink_R_Status_Bit.入库货叉上限检测:=Deliver_In.货叉顶升上限检测;
CCLink_R_Status_Bit.入库货叉下限检测:=Deliver_In.货叉顶升下限检测;
CCLink_R_Status_Bit.入库台上限检测:=Deliver_In.入库口顶升上限检测;
CCLink_R_Status_Bit.入库台下限检测:=Deliver_In.入库口顶升下限检测;
CCLink_R_Status_Bit.出库货叉上限检测:=Deliver_OUT.货叉顶升上限检测;
CCLink_R_Status_Bit.出库货叉下限检测:=Deliver_OUT.货叉顶升下限检测;
CCLink_R_Status_Bit.出库台上限检测:=Deliver_OUT.出库口顶升上限检测;
CCLink_R_Status_Bit.出库台下限检测:=Deliver_OUT.出库口顶升下限检测;
CCLink_R_Status_Bit.入库超宽检测1:=DInput.CV01超宽检测1;
CCLink_R_Status_Bit.入库超宽检测2:=DInput.CV01超宽检测2;
CCLink_R_Status_Bit.入库超高检测:=DInput.CV01超高检测;
CCLink_R_Status_Bit.入库坍塌检测:=DInput.CV01超高检测;
CCLink_R_Status_Bit.入库光栅:=DInput.CV_IN侧安全光栅输入信号1 AND DInput.CV_IN侧安全光栅输入信号2;
CCLink_R_Status_Bit.出库光栅:=DInput.CV_Out侧安全光栅输入信号1 AND DInput.CV_Out侧安全光栅输入信号2;
CCLink_R_Status_Bit.AGV入光栅:=DInput.AGV侧安全光栅输入信号1 AND DInput.AGV侧安全光栅输入信号2;
CCLink_R_Status_Bit.AGV出光栅:=DInput.AGV侧安全光栅输入信号11 AND DInput.AGV侧安全光栅输入信号12;
CCLink_R_Status_Bit.安全门状态:=DInput.安全门1输入信号1 AND DInput.安全门1输入信号2;
CCLink_R_Status_Bit.入库agv本体检测:=Deliver_In.AGV本体检测;
CCLink_R_Status_Bit.入库agv物料检测:=Deliver_In.AGV物料探测;
CCLink_R_Status_Bit.出库agv本体检测:=Deliver_Out.AGV本体检测;
CCLink_R_Status_Bit.出库agv物料检测:=Deliver_Out.AGV物料探测;
CCLink_R_Status_Bit.入库货叉极限:=DInput.CV01伸缩极限检测;
CCLink_R_Status_Bit.入库货叉原点:=DInput.CV01伸缩中位检测1 AND DInput.CV01伸缩中位检测2;
CCLink_R_Status_Bit.出库库货叉极限:=DInput.CV02伸缩极限检测;
CCLink_R_Status_Bit.出库货叉原点:=DInput.CV02伸缩中位检测1 AND DInput.CV02伸缩中位检测2;


(*Write*)

(*Ry*)
END_PROGRAM

FUNCTION_BLOCK I+ST_44a547fe69a44295
VAR_INPUT
  __IST_EN_IN : BOOL;
END_VAR
VAR_OUTPUT
  __IST_EN_OUT : BOOL;
END_VAR
VAR_IN_OUT
  Parse_Done_Cv1 : BOOL;
  RFID1 : INT;
  RFID2 : INT;
  RFID3 : INT;
  RFID4 : INT;
  RFID5 : INT;
  RFID6 : INT;
END_VAR
(* IST HEADER START *)
IF NOT __IST_EN_IN THEN __IST_EN_OUT:=FALSE; RETURN; END_IF;
(* VERSION=1:TYPE=STB *)
(* IST HEADER END *)
IF (U2\G4129 <>RFID1 OR U2\G4130 <>RFID2 OR  U2\G4131 <>RFID3 OR
    U2\G4132 <>RFID4 OR U2\G4133 <>RFID5 OR  U2\G4134 <>RFID6) AND M340=FALSE THEN
    BMOV(1,U2\G4129,6,D600);
    SWAP(1,D600);
    SWAP(1,D601);
    SWAP(1,D602);
    SWAP(1,D603);
    SWAP(1,D604);
    SWAP(1,D605);
    RFID1:=U2\G4129;
    RFID2:=U2\G4130;
    RFID3:=U2\G4131;
    RFID4:=U2\G4132;
    RFID5:=U2\G4133;
    RFID6:=U2\G4134;
END_IF;
IF (U2\G4129 = RFID1 AND U2\G4130 = RFID2 AND  U2\G4131 = RFID3 AND
    U2\G4132 = RFID4 AND U2\G4133 = RFID5 AND  U2\G4134 = RFID6) AND M340=FALSE  THEN
    Parse_Done_Cv1:=TRUE;
END_IF;
END_FUNCTION_BLOCK

FUNCTION_BLOCK I+ST_122ae8440b094ab7
VAR_INPUT
  __IST_EN_IN : BOOL;
END_VAR
VAR_OUTPUT
  __IST_EN_OUT : BOOL;
END_VAR
VAR_IN_OUT
  Parse_Done_Cv2 : BOOL;
  RFID11 : INT;
  RFID12 : INT;
  RFID13 : INT;
  RFID14 : INT;
  RFID15 : INT;
  RFID16 : INT;
END_VAR
(* IST HEADER START *)
IF NOT __IST_EN_IN THEN __IST_EN_OUT:=FALSE; RETURN; END_IF;
(* VERSION=1:TYPE=STB *)
(* IST HEADER END *)
IF (U2\G4193 <>RFID11 OR U2\G4194 <>RFID12 OR  U2\G4195 <>RFID13 OR
    U2\G4196 <>RFID14 OR U2\G4197 <>RFID15 OR  U2\G4198 <>RFID16) AND M341=FALSE THEN
    BMOV(1,U2\G4193,6,D650);
    SWAP(1,D650);
    SWAP(1,D651);
    SWAP(1,D652);
    SWAP(1,D653);
    SWAP(1,D654);
    SWAP(1,D655);
    RFID11:=U2\G4193;
    RFID12:=U2\G4194;
    RFID13:=U2\G4195;
    RFID14:=U2\G4196;
    RFID15:=U2\G4197;
    RFID16:=U2\G4198;
END_IF;
IF (U2\G4193 =RFID11 AND U2\G4194 =RFID12 AND U2\G4195 =RFID13 AND
    U2\G4196 =RFID14 AND U2\G4197 =RFID15 AND U2\G4198 =RFID16) AND M341=FALSE THEN
    Parse_Done_Cv2:=TRUE;
END_IF;
END_FUNCTION_BLOCK
